LIN {X 0,Y 530.47,Z 630.938,A -85,B 0,C 180,E1 -4406.963,E2 -4406.963} C_VEL
LIN {X 0,Y 530.412,Z 632.682,A -85,B 0,C 180,E1 -4407.722,E2 -4407.722} C_VEL
LIN {X 0,Y 530.36,Z 633.93,A -85,B 0,C 180,E1 -4408.482,E2 -4408.482} C_VEL
LIN {X 0,Y 530.342,Z 634.707,A -85,B 0,C 180,E1 -4409.241,E2 -4409.241} C_VEL
LIN {X 0,Y 530.34,Z 635,A -85,B 0,C 180,E1 -4410,E2 -4410} C_VEL
LIN {X 0,Y 530.342,Z 634.706,A -85,B 0,C 180,E1 -4410.76,E2 -4410.76} C_VEL
LIN {X 0,Y 530.36,Z 633.928,A -85,B 0,C 180,E1 -4411.519,E2 -4411.519} C_VEL
LIN {X 0,Y 530.412,Z 632.679,A -85,B 0,C 180,E1 -4412.279,E2 -4412.279} C_VEL
LIN {X 0,Y 530.501,Z 629.785,A -85,B 0,C 180,E1 -4413.418,E2 -4413.418} C_VEL
LIN {X 0,Y 530.546,Z 627.147,A -85,B 0,C 180,E1 -4414.178,E2 -4414.178} C_VEL
LIN {X 0,Y 530.543,Z 621.984,A -85,B 0,C 180,E1 -4415.321,E2 -4415.321} C_VEL
LIN {X 0,Y 530.729,Z 616.44,A -85,B 0,C 180,E1 -4416.271,E2 -4416.271} C_VEL
LIN {X 0,Y 530.794,Z 609.432,A -85,B 0,C 180,E1 -4417.226,E2 -4417.226} C_VEL
LIN {X 0,Y 530.928,Z 601.415,A -85,B 0,C 180,E1 -4418.086,E2 -4418.086} C_VEL
LIN {X 0,Y 531.106,Z 593.759,A -85,B 0,C 180,E1 -4418.753,E2 -4418.753} C_VEL
LIN {X 0,Y 531.226,Z 585.716,A -85,B 0,C 180,E1 -4419.327,E2 -4419.327} C_VEL
LIN {X 0,Y 531.389,Z 577.382,A -85,B 0,C 180,E1 -4419.805,E2 -4419.805} C_VEL
LIN {X 0,Y 531.523,Z 568.876,A -85,B 0,C 180,E1 -4420.187,E2 -4420.187} C_VEL
LIN {X 0,Y 531.454,Z 560.399,A -85,B 0,C 180,E1 -4420.477,E2 -4420.477} C_VEL
LIN {X 0,Y 530.57,Z 553.301,A -85,B 0,C 180,E1 -4420.688,E2 -4420.688} C_VEL
LIN {X 0,Y 530.658,Z 544.2,A -85,B 0,C 180,E1 -4423.402,E2 -4423.402} C_VEL
LIN {X 0,Y 530.751,Z 534.941,A -85,B 0,C 180,E1 -4426.146,E2 -4426.146} C_VEL
LIN {X 0,Y 530.856,Z 525.622,A -85,B 0,C 180,E1 -4428.927,E2 -4428.927} C_VEL
LIN {X 0,Y 530.984,Z 515.377,A -85,B 0,C 180,E1 -4432.104,E2 -4432.104} C_VEL
LIN {X 0,Y 531.159,Z 506.089,A -85,B 0,C 180,E1 -4435.05,E2 -4435.05} C_VEL
LIN {X 0,Y 531.329,Z 497.227,A -85,B 0,C 180,E1 -4438.006,E2 -4438.006} C_VEL
LIN {X 0,Y 531.612,Z 488.788,A -85,B 0,C 180,E1 -4441.037,E2 -4441.037} C_VEL
LIN {X 0,Y 531.787,Z 484.27,A -85,B 0,C 180,E1 -4442.81,E2 -4442.81} C_VEL
LIN {X 0,Y 530.978,Z 479.161,A -85,B 0,C 180,E1 -4445.126,E2 -4445.126} C_VEL
LIN {X 0,Y 530.969,Z 479.161,A -85,B 0,C 180,E1 -4447.508,E2 -4447.508} C_VEL
LIN {X 0,Y 530.986,Z 479.159,A -85,B 0,C 180,E1 -4450.433,E2 -4450.433} C_VEL
LIN {X 0,Y 530.968,Z 479.162,A -85,B 0,C 180,E1 -4453.495,E2 -4453.495} C_VEL
LIN {X 0,Y 530.97,Z 479.161,A -85,B 0,C 180,E1 -4456.506,E2 -4456.506} C_VEL
LIN {X 0,Y 530.984,Z 479.159,A -85,B 0,C 180,E1 -4459.567,E2 -4459.567} C_VEL
LIN {X 0,Y 530.971,Z 479.159,A -85,B 0,C 180,E1 -4462.577,E2 -4462.577} C_VEL
LIN {X 0,Y 530.985,Z 479.156,A -85,B 0,C 180,E1 -4465.31,E2 -4465.31} C_VEL
LIN {X 0,Y 530.889,Z 479.172,A -85,B 0,C 180,E1 -4468.027,E2 -4468.027} C_VEL
LIN {X 0,Y 530.823,Z 481.04,A -85,B 0,C 180,E1 -4469.794,E2 -4469.794} C_VEL
LIN {X 0,Y 530.741,Z 484.422,A -85,B 0,C 180,E1 -4472.525,E2 -4472.525} C_VEL
LIN {X 0,Y 530.652,Z 487.475,A -85,B 0,C 180,E1 -4474.925,E2 -4474.925} C_VEL
LIN {X 0,Y 530.59,Z 490.671,A -85,B 0,C 180,E1 -4477.411,E2 -4477.411} C_VEL
LIN {X 0,Y 530.592,Z 494.26,A -85,B 0,C 180,E1 -4480.126,E2 -4480.126} C_VEL
LIN {X 0,Y 530.52,Z 498.183,A -85,B 0,C 180,E1 -4483.056,E2 -4483.056} C_VEL
LIN {X 0,Y 530.533,Z 501.331,A -85,B 0,C 180,E1 -4485.422,E2 -4485.422} C_VEL
LIN {X 0,Y 530.451,Z 505.76,A -85,B 0,C 180,E1 -4488.649,E2 -4488.649} C_VEL
LIN {X 0,Y 530.428,Z 506.855,A -85,B 0,C 180,E1 -4489.431,E2 -4489.431} C_VEL
LIN {X 0,Y 531.541,Z 516.565,A -85,B 0,C 180,E1 -4489.766,E2 -4489.766} C_VEL
LIN {X 0,Y 531.394,Z 526.519,A -85,B 0,C 180,E1 -4490.196,E2 -4490.196} C_VEL
LIN {X 0,Y 531.236,Z 535.019,A -85,B 0,C 180,E1 -4490.673,E2 -4490.673} C_VEL
LIN {X 0,Y 531.105,Z 543.186,A -85,B 0,C 180,E1 -4491.247,E2 -4491.247} C_VEL
LIN {X 0,Y 530.929,Z 550.939,A -85,B 0,C 180,E1 -4491.915,E2 -4491.915} C_VEL
LIN {X 0,Y 530.797,Z 559.04,A -85,B 0,C 180,E1 -4492.774,E2 -4492.774} C_VEL
LIN {X 0,Y 530.739,Z 566.143,A -85,B 0,C 180,E1 -4493.726,E2 -4493.726} C_VEL
LIN {X 0,Y 530.544,Z 571.76,A -85,B 0,C 180,E1 -4494.68,E2 -4494.68} C_VEL
LIN {X 0,Y 530.547,Z 576.97,A -85,B 0,C 180,E1 -4495.822,E2 -4495.822} C_VEL
LIN {X 0,Y 530.503,Z 579.65,A -85,B 0,C 180,E1 -4496.582,E2 -4496.582} C_VEL
LIN {X 0,Y 530.411,Z 582.584,A -85,B 0,C 180,E1 -4497.722,E2 -4497.722} C_VEL
LIN {X 0,Y 530.361,Z 583.871,A -85,B 0,C 180,E1 -4498.481,E2 -4498.481} C_VEL
LIN {X 0,Y 530.341,Z 584.687,A -85,B 0,C 180,E1 -4499.241,E2 -4499.241} C_VEL
LIN {X 0,Y 530.339,Z 584.997,A -85,B 0,C 180,E1 -4500,E2 -4500} C_VEL
LIN {X 0,Y 530.343,Z 584.725,A -85,B 0,C 180,E1 -4500.759,E2 -4500.759} C_VEL
LIN {X 0,Y 530.36,Z 583.986,A -85,B 0,C 180,E1 -4501.519,E2 -4501.519} C_VEL
LIN {X 0,Y 530.411,Z 582.776,A -85,B 0,C 180,E1 -4502.278,E2 -4502.278} C_VEL
LIN {X 0,Y 530.491,Z 579.923,A -85,B 0,C 180,E1 -4503.418,E2 -4503.418} C_VEL
LIN {X 0,Y 530.546,Z 577.328,A -85,B 0,C 180,E1 -4504.178,E2 -4504.178} C_VEL
LIN {X 0,Y 530.541,Z 572.214,A -85,B 0,C 180,E1 -4505.321,E2 -4505.321} C_VEL
LIN {X 0,Y 530.729,Z 566.748,A -85,B 0,C 180,E1 -4506.266,E2 -4506.266} C_VEL
LIN {X 0,Y 530.795,Z 559.812,A -85,B 0,C 180,E1 -4507.226,E2 -4507.226} C_VEL
LIN {X 0,Y 530.918,Z 551.89,A -85,B 0,C 180,E1 -4508.085,E2 -4508.085} C_VEL
LIN {X 0,Y 531.092,Z 544.335,A -85,B 0,C 180,E1 -4508.753,E2 -4508.753} C_VEL
LIN {X 0,Y 531.22,Z 536.423,A -85,B 0,C 180,E1 -4509.327,E2 -4509.327} C_VEL
LIN {X 0,Y 531.392,Z 528.262,A -85,B 0,C 180,E1 -4509.804,E2 -4509.804} C_VEL
LIN {X 0,Y 531.484,Z 520.02,A -85,B 0,C 180,E1 -4510.187,E2 -4510.187} C_VEL
LIN {X 0,Y 531.275,Z 513.221,A -85,B 0,C 180,E1 -4510.444,E2 -4510.444} C_VEL
LIN {X 0,Y 530.419,Z 506.574,A -85,B 0,C 180,E1 -4510.666,E2 -4510.666} C_VEL
LIN {X 0,Y 530.455,Z 502.979,A -85,B 0,C 180,E1 -4513.017,E2 -4513.017} C_VEL
LIN {X 0,Y 530.498,Z 499.448,A -85,B 0,C 180,E1 -4515.365,E2 -4515.365} C_VEL
LIN {X 0,Y 530.51,Z 495.947,A -85,B 0,C 180,E1 -4517.74,E2 -4517.74} C_VEL
LIN {X 0,Y 530.574,Z 492.447,A -85,B 0,C 180,E1 -4520.145,E2 -4520.145} C_VEL
LIN {X 0,Y 530.535,Z 488.732,A -85,B 0,C 180,E1 -4522.592,E2 -4522.592} C_VEL
LIN {X 0,Y 530.602,Z 485.059,A -85,B 0,C 180,E1 -4525.078,E2 -4525.078} C_VEL
LIN {X 0,Y 530.739,Z 481.892,A -85,B 0,C 180,E1 -4527.292,E2 -4527.292} C_VEL
LIN {X 0,Y 530.746,Z 488.059,A -85,B 0,C 180,E1 -4529.773,E2 -4529.773} C_VEL
LIN {X 0,Y 530.77,Z 494.522,A -85,B 0,C 180,E1 -4532.439,E2 -4532.439} C_VEL
LIN {X 0,Y 530.667,Z 500.16,A -85,B 0,C 180,E1 -4534.803,E2 -4534.803} C_VEL
LIN {X 0,Y 530.626,Z 506.621,A -85,B 0,C 180,E1 -4537.536,E2 -4537.536} C_VEL
LIN {X 0,Y 530.597,Z 511.429,A -85,B 0,C 180,E1 -4539.542,E2 -4539.542} C_VEL
LIN {X 0,Y 529.942,Z 512.958,A -85,B 0,C 180,E1 -4540.154,E2 -4540.154} C_VEL
LIN {X 0,Y 527.033,Z 515.502,A -85,B 0,C 180,E1 -4541.145,E2 -4541.145} C_VEL
LIN {X 0,Y 524.569,Z 517.514,A -85,B 0,C 180,E1 -4541.944,E2 -4541.944} C_VEL
LIN {X 0,Y 523.523,Z 518.992,A -85,B 0,C 180,E1 -4542.563,E2 -4542.563} C_VEL
LIN {X 0,Y 523.447,Z 519.474,A -85,B 0,C 180,E1 -4542.773,E2 -4542.773} C_VEL
LIN {X 0,Y 523.418,Z 525.143,A -85,B 0,C 180,E1 -4545.254,E2 -4545.254} C_VEL
LIN {X 0,Y 524.584,Z 535.182,A -85,B 0,C 180,E1 -4545.573,E2 -4545.573} C_VEL
LIN {X 0,Y 524.442,Z 546.72,A -85,B 0,C 180,E1 -4546.064,E2 -4546.064} C_VEL
LIN {X 0,Y 524.216,Z 556.215,A -85,B 0,C 180,E1 -4546.615,E2 -4546.615} C_VEL
LIN {X 0,Y 524.055,Z 564.577,A -85,B 0,C 180,E1 -4547.23,E2 -4547.23} C_VEL
LIN {X 0,Y 523.854,Z 572.859,A -85,B 0,C 180,E1 -4547.987,E2 -4547.987} C_VEL
LIN {X 0,Y 523.695,Z 579.437,A -85,B 0,C 180,E1 -4548.722,E2 -4548.722} C_VEL
LIN {X 0,Y 523.595,Z 584.439,A -85,B 0,C 180,E1 -4549.383,E2 -4549.383} C_VEL
LIN {X 0,Y 523.513,Z 590.665,A -85,B 0,C 180,E1 -4550.399,E2 -4550.399} C_VEL
LIN {X 0,Y 523.446,Z 594.425,A -85,B 0,C 180,E1 -4551.145,E2 -4551.145} C_VEL
LIN {X 0,Y 523.416,Z 597.403,A -85,B 0,C 180,E1 -4551.855,E2 -4551.855} C_VEL
LIN {X 0,Y 523.337,Z 600.555,A -85,B 0,C 180,E1 -4552.82,E2 -4552.82} C_VEL
LIN {X 0,Y 523.282,Z 602.795,A -85,B 0,C 180,E1 -4553.775,E2 -4553.775} C_VEL
LIN {X 0,Y 523.279,Z 604.553,A -85,B 0,C 180,E1 -4555.012,E2 -4555.012} C_VEL
LIN {X 0,Y 523.279,Z 604.883,A -85,B 0,C 180,E1 -4556.377,E2 -4556.377} C_VEL
LIN {X 0,Y 523.278,Z 603.641,A -85,B 0,C 180,E1 -4557.794,E2 -4557.794} C_VEL
LIN {X 0,Y 523.31,Z 602.57,A -85,B 0,C 180,E1 -4558.414,E2 -4558.414} C_VEL
LIN {X 0,Y 523.392,Z 600.399,A -85,B 0,C 180,E1 -4559.319,E2 -4559.319} C_VEL
LIN {X 0,Y 523.42,Z 596.195,A -85,B 0,C 180,E1 -4560.525,E2 -4560.525} C_VEL
LIN {X 0,Y 523.454,Z 592.668,A -85,B 0,C 180,E1 -4561.315,E2 -4561.315} C_VEL
LIN {X 0,Y 523.556,Z 587.76,A -85,B 0,C 180,E1 -4562.201,E2 -4562.201} C_VEL
LIN {X 0,Y 523.668,Z 581.842,A -85,B 0,C 180,E1 -4563.067,E2 -4563.067} C_VEL
LIN {X 0,Y 523.803,Z 574.832,A -85,B 0,C 180,E1 -4563.9,E2 -4563.9} C_VEL
LIN {X 0,Y 523.945,Z 567.889,A -85,B 0,C 180,E1 -4564.581,E2 -4564.581} C_VEL
LIN {X 0,Y 524.142,Z 559.814,A -85,B 0,C 180,E1 -4565.227,E2 -4565.227} C_VEL
LIN {X 0,Y 524.261,Z 550.824,A -85,B 0,C 180,E1 -4565.803,E2 -4565.803} C_VEL
LIN {X 0,Y 524.478,Z 541.798,A -85,B 0,C 180,E1 -4566.253,E2 -4566.253} C_VEL
LIN {X 0,Y 524.415,Z 533.272,A -85,B 0,C 180,E1 -4566.581,E2 -4566.581} C_VEL
LIN {X 0,Y 523.368,Z 525.332,A -85,B 0,C 180,E1 -4566.846,E2 -4566.846} C_VEL
LIN {X 0,Y 523.456,Z 518.488,A -85,B 0,C 180,E1 -4570.023,E2 -4570.023} C_VEL
LIN {X 0,Y 523.489,Z 512.468,A -85,B 0,C 180,E1 -4572.821,E2 -4572.821} C_VEL
LIN {X 0,Y 523.565,Z 505.401,A -85,B 0,C 180,E1 -4576.017,E2 -4576.017} C_VEL
LIN {X 0,Y 523.665,Z 498.515,A -85,B 0,C 180,E1 -4579.17,E2 -4579.17} C_VEL
LIN {X 0,Y 523.664,Z 491.614,A -85,B 0,C 180,E1 -4582.287,E2 -4582.287} C_VEL
LIN {X 0,Y 523.761,Z 484.698,A -85,B 0,C 180,E1 -4585.382,E2 -4585.382} C_VEL
LIN {X 0,Y 523.697,Z 480.067,A -85,B 0,C 180,E1 -4587.5,E2 -4587.5} C_VEL
LIN {X 0,Y 524.123,Z 480.013,A -85,B 0,C 180,E1 -4589.231,E2 -4589.231} C_VEL
LIN {X 0,Y 524.115,Z 480.013,A -85,B 0,C 180,E1 -4592.305,E2 -4592.305} C_VEL
LIN {X 0,Y 524.087,Z 480.017,A -85,B 0,C 180,E1 -4595.386,E2 -4595.386} C_VEL
LIN {X 0,Y 524.003,Z 480.028,A -85,B 0,C 180,E1 -4598.484,E2 -4598.484} C_VEL
LIN {X 0,Y 524.004,Z 480.026,A -85,B 0,C 180,E1 -4601.739,E2 -4601.739} C_VEL
LIN {X 0,Y 523.995,Z 480.027,A -85,B 0,C 180,E1 -4605.052,E2 -4605.052} C_VEL
LIN {X 0,Y 523.966,Z 480.032,A -85,B 0,C 180,E1 -4607.968,E2 -4607.968} C_VEL
LIN {X 0,Y 523.973,Z 480.032,A -85,B 0,C 180,E1 -4610.41,E2 -4610.41} C_VEL
LIN {X 0,Y 523.918,Z 480.039,A -85,B 0,C 180,E1 -4612.893,E2 -4612.893} C_VEL
LIN {X 0,Y 523.956,Z 480.034,A -85,B 0,C 180,E1 -4615.418,E2 -4615.418} C_VEL
LIN {X 0,Y 523.971,Z 480.032,A -85,B 0,C 180,E1 -4617.998,E2 -4617.998} C_VEL
LIN {X 0,Y 523.953,Z 480.033,A -85,B 0,C 180,E1 -4620.856,E2 -4620.856} C_VEL
LIN {X 0,Y 523.961,Z 480.034,A -85,B 0,C 180,E1 -4623.735,E2 -4623.735} C_VEL
LIN {X 0,Y 523.923,Z 480.037,A -85,B 0,C 180,E1 -4626.404,E2 -4626.404} C_VEL
LIN {X 0,Y 523.922,Z 480.036,A -85,B 0,C 180,E1 -4629.084,E2 -4629.084} C_VEL
LIN {X 0,Y 523.953,Z 480.034,A -85,B 0,C 180,E1 -4632.118,E2 -4632.118} C_VEL
LIN {X 0,Y 523.955,Z 480.033,A -85,B 0,C 180,E1 -4635.308,E2 -4635.308} C_VEL
LIN {X 0,Y 523.973,Z 480.031,A -85,B 0,C 180,E1 -4638.687,E2 -4638.687} C_VEL
LIN {X 0,Y 523.952,Z 480.033,A -85,B 0,C 180,E1 -4641.075,E2 -4641.075} C_VEL
LIN {X 0,Y 523.898,Z 480.042,A -85,B 0,C 180,E1 -4643.825,E2 -4643.825} C_VEL
LIN {X 0,Y 523.94,Z 480.034,A -85,B 0,C 180,E1 -4646.635,E2 -4646.635} C_VEL
LIN {X 0,Y 523.955,Z 480.032,A -85,B 0,C 180,E1 -4649.356,E2 -4649.356} C_VEL
LIN {X 0,Y 523.979,Z 480.03,A -85,B 0,C 180,E1 -4652.28,E2 -4652.28} C_VEL
LIN {X 0,Y 523.954,Z 480.032,A -85,B 0,C 180,E1 -4654.581,E2 -4654.581} C_VEL
LIN {X 0,Y 523.915,Z 480.037,A -85,B 0,C 180,E1 -4657.107,E2 -4657.107} C_VEL
LIN {X 0,Y 523.978,Z 480.03,A -85,B 0,C 180,E1 -4659.865,E2 -4659.865} C_VEL
LIN {X 0,Y 523.965,Z 480.032,A -85,B 0,C 180,E1 -4662.837,E2 -4662.837} C_VEL
LIN {X 0,Y 523.975,Z 480.031,A -85,B 0,C 180,E1 -4665.236,E2 -4665.236} C_VEL
LIN {X 0,Y 524.013,Z 480.028,A -85,B 0,C 180,E1 -4668.394,E2 -4668.394} C_VEL
LIN {X 0,Y 524.003,Z 480.027,A -85,B 0,C 180,E1 -4671.516,E2 -4671.516} C_VEL
LIN {X 0,Y 524.081,Z 480.017,A -85,B 0,C 180,E1 -4674.614,E2 -4674.614} C_VEL
LIN {X 0,Y 524.112,Z 480.014,A -85,B 0,C 180,E1 -4677.694,E2 -4677.694} C_VEL
LIN {X 0,Y 524.122,Z 480.011,A -85,B 0,C 180,E1 -4680.768,E2 -4680.768} C_VEL
LIN {X 0,Y 524.074,Z 480.018,A -85,B 0,C 180,E1 -4683.075,E2 -4683.075} C_VEL
LIN {X 0,Y 524.046,Z 480.024,A -85,B 0,C 180,E1 -4686.159,E2 -4686.159} C_VEL
LIN {X 0,Y 523.999,Z 480.027,A -85,B 0,C 180,E1 -4689.262,E2 -4689.262} C_VEL
LIN {X 0,Y 524.001,Z 480.027,A -85,B 0,C 180,E1 -4691.74,E2 -4691.74} C_VEL
LIN {X 0,Y 523.99,Z 480.028,A -85,B 0,C 180,E1 -4695.052,E2 -4695.052} C_VEL
LIN {X 0,Y 523.962,Z 480.034,A -85,B 0,C 180,E1 -4697.969,E2 -4697.969} C_VEL
LIN {X 0,Y 523.97,Z 480.032,A -85,B 0,C 180,E1 -4700.41,E2 -4700.41} C_VEL
LIN {X 0,Y 523.915,Z 480.039,A -85,B 0,C 180,E1 -4702.893,E2 -4702.893} C_VEL
LIN {X 0,Y 523.951,Z 480.034,A -85,B 0,C 180,E1 -4705.419,E2 -4705.419} C_VEL
LIN {X 0,Y 523.967,Z 480.031,A -85,B 0,C 180,E1 -4707.999,E2 -4707.999} C_VEL
LIN {X 0,Y 523.951,Z 480.033,A -85,B 0,C 180,E1 -4710.857,E2 -4710.857} C_VEL
LIN {X 0,Y 523.959,Z 480.033,A -85,B 0,C 180,E1 -4713.735,E2 -4713.735} C_VEL
LIN {X 0,Y 523.921,Z 480.036,A -85,B 0,C 180,E1 -4716.405,E2 -4716.405} C_VEL
LIN {X 0,Y 523.918,Z 480.038,A -85,B 0,C 180,E1 -4719.085,E2 -4719.085} C_VEL
LIN {X 0,Y 523.956,Z 480.032,A -85,B 0,C 180,E1 -4722.118,E2 -4722.118} C_VEL
LIN {X 0,Y 523.953,Z 480.035,A -85,B 0,C 180,E1 -4725.309,E2 -4725.309} C_VEL
LIN {X 0,Y 523.971,Z 480.032,A -85,B 0,C 180,E1 -4728.688,E2 -4728.688} C_VEL
LIN {X 0,Y 523.952,Z 480.035,A -85,B 0,C 180,E1 -4731.076,E2 -4731.076} C_VEL
LIN {X 0,Y 523.927,Z 480.037,A -85,B 0,C 180,E1 -4733.828,E2 -4733.828} C_VEL
LIN {X 0,Y 523.978,Z 480.097,A -85,B 0,C 180,E1 -4736.868,E2 -4736.868} C_VEL
LIN {X 0,Y 524.761,Z 484.749,A -85,B 0,C 180,E1 -4738.513,E2 -4738.513} C_VEL
LIN {X 0,Y 524.676,Z 490.829,A -85,B 0,C 180,E1 -4740.537,E2 -4740.537} C_VEL
LIN {X 0,Y 524.437,Z 499.476,A -85,B 0,C 180,E1 -4743.325,E2 -4743.325} C_VEL
LIN {X 0,Y 524.185,Z 508.922,A -85,B 0,C 180,E1 -4746.283,E2 -4746.283} C_VEL
LIN {X 0,Y 524.034,Z 518.43,A -85,B 0,C 180,E1 -4749.182,E2 -4749.182} C_VEL
LIN {X 0,Y 523.812,Z 528.83,A -85,B 0,C 180,E1 -4752.29,E2 -4752.29} C_VEL
LIN {X 0,Y 523.702,Z 539.019,A -85,B 0,C 180,E1 -4755.228,E2 -4755.228} C_VEL
LIN {X 0,Y 523.603,Z 550.38,A -85,B 0,C 180,E1 -4758.473,E2 -4758.473} C_VEL
LIN {X 0,Y 523.549,Z 552.826,A -85,B 0,C 180,E1 -4759.168,E2 -4759.168} C_VEL
LIN {X 0,Y 524.574,Z 563.488,A -85,B 0,C 180,E1 -4759.483,E2 -4759.483} C_VEL
LIN {X 0,Y 524.423,Z 575.323,A -85,B 0,C 180,E1 -4759.967,E2 -4759.967} C_VEL
LIN {X 0,Y 524.232,Z 584.068,A -85,B 0,C 180,E1 -4760.451,E2 -4760.451} C_VEL
LIN {X 0,Y 524.122,Z 592.427,A -85,B 0,C 180,E1 -4761.033,E2 -4761.033} C_VEL
LIN {X 0,Y 523.923,Z 600.332,A -85,B 0,C 180,E1 -4761.709,E2 -4761.709} C_VEL
LIN {X 0,Y 523.757,Z 607.725,A -85,B 0,C 180,E1 -4762.483,E2 -4762.483} C_VEL
LIN {X 0,Y 523.659,Z 615.797,A -85,B 0,C 180,E1 -4763.54,E2 -4763.54} C_VEL
LIN {X 0,Y 523.485,Z 621.991,A -85,B 0,C 180,E1 -4764.608,E2 -4764.608} C_VEL
LIN {X 0,Y 523.472,Z 627.151,A -85,B 0,C 180,E1 -4765.766,E2 -4765.766} C_VEL
LIN {X 0,Y 523.381,Z 630.939,A -85,B 0,C 180,E1 -4766.921,E2 -4766.921} C_VEL
LIN {X 0,Y 523.336,Z 632.681,A -85,B 0,C 180,E1 -4767.691,E2 -4767.691} C_VEL
LIN {X 0,Y 523.273,Z 633.929,A -85,B 0,C 180,E1 -4768.461,E2 -4768.461} C_VEL
LIN {X 0,Y 523.248,Z 634.706,A -85,B 0,C 180,E1 -4769.231,E2 -4769.231} C_VEL
LIN {X 0,Y 523.244,Z 635,A -85,B 0,C 180,E1 -4770,E2 -4770} C_VEL
LIN {X 0,Y 523.248,Z 634.705,A -85,B 0,C 180,E1 -4770.77,E2 -4770.77} C_VEL
LIN {X 0,Y 523.273,Z 633.927,A -85,B 0,C 180,E1 -4771.54,E2 -4771.54} C_VEL
LIN {X 0,Y 523.336,Z 632.678,A -85,B 0,C 180,E1 -4772.309,E2 -4772.309} C_VEL
LIN {X 0,Y 523.413,Z 629.785,A -85,B 0,C 180,E1 -4773.464,E2 -4773.464} C_VEL
LIN {X 0,Y 523.47,Z 627.147,A -85,B 0,C 180,E1 -4774.235,E2 -4774.235} C_VEL
LIN {X 0,Y 523.485,Z 621.984,A -85,B 0,C 180,E1 -4775.393,E2 -4775.393} C_VEL
LIN {X 0,Y 523.668,Z 615.737,A -85,B 0,C 180,E1 -4776.469,E2 -4776.469} C_VEL
LIN {X 0,Y 523.758,Z 607.72,A -85,B 0,C 180,E1 -4777.518,E2 -4777.518} C_VEL
LIN {X 0,Y 523.924,Z 600.325,A -85,B 0,C 180,E1 -4778.291,E2 -4778.291} C_VEL
LIN {X 0,Y 524.123,Z 592.401,A -85,B 0,C 180,E1 -4778.968,E2 -4778.968} C_VEL
LIN {X 0,Y 524.243,Z 584.023,A -85,B 0,C 180,E1 -4779.55,E2 -4779.55} C_VEL
LIN {X 0,Y 524.459,Z 573.336,A -85,B 0,C 180,E1 -4780.13,E2 -4780.13} C_VEL
LIN {X 0,Y 524.584,Z 562.538,A -85,B 0,C 180,E1 -4780.542,E2 -4780.542} C_VEL
LIN {X 0,Y 523.502,Z 553.04,A -85,B 0,C 180,E1 -4780.834,E2 -4780.834} C_VEL
LIN {X 0,Y 523.601,Z 542.52,A -85,B 0,C 180,E1 -4783.982,E2 -4783.982} C_VEL
LIN {X 0,Y 523.688,Z 533.247,A -85,B 0,C 180,E1 -4786.771,E2 -4786.771} C_VEL
LIN {X 0,Y 523.834,Z 524.034,A -85,B 0,C 180,E1 -4789.598,E2 -4789.598} C_VEL
LIN {X 0,Y 523.992,Z 513.633,A -85,B 0,C 180,E1 -4792.89,E2 -4792.89} C_VEL
LIN {X 0,Y 524.182,Z 503.917,A -85,B 0,C 180,E1 -4796.064,E2 -4796.064} C_VEL
LIN {X 0,Y 524.39,Z 495.936,A -85,B 0,C 180,E1 -4798.848,E2 -4798.848} C_VEL
LIN {X 0,Y 524.683,Z 488.876,A -85,B 0,C 180,E1 -4801.493,E2 -4801.493} C_VEL
LIN {X 0,Y 524.82,Z 486.443,A -85,B 0,C 180,E1 -4802.473,E2 -4802.473} C_VEL
LIN {X 0,Y 524.412,Z 482.418,A -85,B 0,C 180,E1 -4804.255,E2 -4804.255} C_VEL
LIN {X 0,Y 523.936,Z 480.038,A -85,B 0,C 180,E1 -4805.461,E2 -4805.461} C_VEL
LIN {X 0,Y 523.919,Z 480.039,A -85,B 0,C 180,E1 -4808.102,E2 -4808.102} C_VEL
LIN {X 0,Y 523.944,Z 480.034,A -85,B 0,C 180,E1 -4811.092,E2 -4811.092} C_VEL
LIN {X 0,Y 523.944,Z 480.033,A -85,B 0,C 180,E1 -4814.228,E2 -4814.228} C_VEL
LIN {X 0,Y 523.928,Z 480.038,A -85,B 0,C 180,E1 -4816.834,E2 -4816.834} C_VEL
LIN {X 0,Y 523.944,Z 480.033,A -85,B 0,C 180,E1 -4818.908,E2 -4818.908} C_VEL
LIN {X 0,Y 523.918,Z 480.037,A -85,B 0,C 180,E1 -4821.898,E2 -4821.898} C_VEL
LIN {X 0,Y 523.927,Z 480.038,A -85,B 0,C 180,E1 -4824.911,E2 -4824.911} C_VEL
LIN {X 0,Y 523.871,Z 480.046,A -85,B 0,C 180,E1 -4827.692,E2 -4827.692} C_VEL
LIN {X 0,Y 523.819,Z 480.37,A -85,B 0,C 180,E1 -4828.449,E2 -4828.449} C_VEL
LIN {X 0,Y 523.713,Z 483.539,A -85,B 0,C 180,E1 -4831.112,E2 -4831.112} C_VEL
LIN {X 0,Y 523.654,Z 487.162,A -85,B 0,C 180,E1 -4834.055,E2 -4834.055} C_VEL
LIN {X 0,Y 523.584,Z 489.932,A -85,B 0,C 180,E1 -4836.254,E2 -4836.254} C_VEL
LIN {X 0,Y 523.532,Z 494.212,A -85,B 0,C 180,E1 -4839.572,E2 -4839.572} C_VEL
LIN {X 0,Y 523.445,Z 498.554,A -85,B 0,C 180,E1 -4842.82,E2 -4842.82} C_VEL
LIN {X 0,Y 523.465,Z 501.697,A -85,B 0,C 180,E1 -4845.221,E2 -4845.221} C_VEL
LIN {X 0,Y 523.399,Z 506.246,A -85,B 0,C 180,E1 -4848.586,E2 -4848.586} C_VEL
LIN {X 0,Y 523.388,Z 507.452,A -85,B 0,C 180,E1 -4849.311,E2 -4849.311} C_VEL
LIN {X 0,Y 524.547,Z 516.773,A -85,B 0,C 180,E1 -4849.628,E2 -4849.628} C_VEL
LIN {X 0,Y 524.405,Z 526.74,A -85,B 0,C 180,E1 -4850.064,E2 -4850.064} C_VEL
LIN {X 0,Y 524.238,Z 535.245,A -85,B 0,C 180,E1 -4850.548,E2 -4850.548} C_VEL
LIN {X 0,Y 524.094,Z 543.404,A -85,B 0,C 180,E1 -4851.129,E2 -4851.129} C_VEL
LIN {X 0,Y 523.918,Z 551.144,A -85,B 0,C 180,E1 -4851.806,E2 -4851.806} C_VEL
LIN {X 0,Y 523.761,Z 557.531,A -85,B 0,C 180,E1 -4852.483,E2 -4852.483} C_VEL
LIN {X 0,Y 523.672,Z 563.785,A -85,B 0,C 180,E1 -4853.281,E2 -4853.281} C_VEL
LIN {X 0,Y 523.547,Z 570.93,A -85,B 0,C 180,E1 -4854.415,E2 -4854.415} C_VEL
LIN {X 0,Y 523.422,Z 575.568,A -85,B 0,C 180,E1 -4855.379,E2 -4855.379} C_VEL
LIN {X 0,Y 523.459,Z 578.555,A -85,B 0,C 180,E1 -4856.151,E2 -4856.151} C_VEL
LIN {X 0,Y 523.384,Z 580.875,A -85,B 0,C 180,E1 -4856.921,E2 -4856.921} C_VEL
LIN {X 0,Y 523.336,Z 582.646,A -85,B 0,C 180,E1 -4857.691,E2 -4857.691} C_VEL
LIN {X 0,Y 523.275,Z 583.925,A -85,B 0,C 180,E1 -4858.461,E2 -4858.461} C_VEL
LIN {X 0,Y 523.248,Z 584.735,A -85,B 0,C 180,E1 -4859.23,E2 -4859.23} C_VEL
LIN {X 0,Y 523.243,Z 585.042,A -85,B 0,C 180,E1 -4860,E2 -4860} C_VEL
LIN {X 0,Y 523.249,Z 584.771,A -85,B 0,C 180,E1 -4860.77,E2 -4860.77} C_VEL
LIN {X 0,Y 523.274,Z 584.035,A -85,B 0,C 180,E1 -4861.539,E2 -4861.539} C_VEL
LIN {X 0,Y 523.335,Z 582.831,A -85,B 0,C 180,E1 -4862.309,E2 -4862.309} C_VEL
LIN {X 0,Y 523.404,Z 579.994,A -85,B 0,C 180,E1 -4863.464,E2 -4863.464} C_VEL
LIN {X 0,Y 523.469,Z 577.412,A -85,B 0,C 180,E1 -4864.235,E2 -4864.235} C_VEL
LIN {X 0,Y 523.485,Z 572.326,A -85,B 0,C 180,E1 -4865.393,E2 -4865.393} C_VEL
LIN {X 0,Y 523.643,Z 568.01,A -85,B 0,C 180,E1 -4866.164,E2 -4866.164} C_VEL
LIN {X 0,Y 523.704,Z 561.42,A -85,B 0,C 180,E1 -4867.131,E2 -4867.131} C_VEL
LIN {X 0,Y 523.853,Z 553.062,A -85,B 0,C 180,E1 -4868.098,E2 -4868.098} C_VEL
LIN {X 0,Y 524.089,Z 544.491,A -85,B 0,C 180,E1 -4868.871,E2 -4868.871} C_VEL
LIN {X 0,Y 524.232,Z 536.576,A -85,B 0,C 180,E1 -4869.452,E2 -4869.452} C_VEL
LIN {X 0,Y 524.408,Z 528.402,A -85,B 0,C 180,E1 -4869.936,E2 -4869.936} C_VEL
LIN {X 0,Y 524.507,Z 520.13,A -85,B 0,C 180,E1 -4870.324,E2 -4870.324} C_VEL
LIN {X 0,Y 524.461,Z 515.259,A -85,B 0,C 180,E1 -4870.52,E2 -4870.52} C_VEL
LIN {X 0,Y 523.353,Z 506.81,A -85,B 0,C 180,E1 -4870.812,E2 -4870.812} C_VEL
LIN {X 0,Y 523.365,Z 503.202,A -85,B 0,C 180,E1 -4873.196,E2 -4873.196} C_VEL
LIN {X 0,Y 523.41,Z 499.674,A -85,B 0,C 180,E1 -4875.578,E2 -4875.578} C_VEL
LIN {X 0,Y 523.423,Z 496.175,A -85,B 0,C 180,E1 -4877.988,E2 -4877.988} C_VEL
LIN {X 0,Y 523.482,Z 492.502,A -85,B 0,C 180,E1 -4880.43,E2 -4880.43} C_VEL
LIN {X 0,Y 523.539,Z 487.616,A -85,B 0,C 180,E1 -4883.748,E2 -4883.748} C_VEL
LIN {X 0,Y 523.567,Z 483.933,A -85,B 0,C 180,E1 -4886.294,E2 -4886.294} C_VEL
LIN {X 0,Y 523.693,Z 482.66,A -85,B 0,C 180,E1 -4887.311,E2 -4887.311} C_VEL
LIN {X 0,Y 523.666,Z 488.633,A -85,B 0,C 180,E1 -4889.773,E2 -4889.773} C_VEL
LIN {X 0,Y 523.699,Z 495.221,A -85,B 0,C 180,E1 -4892.466,E2 -4892.466} C_VEL
LIN {X 0,Y 523.58,Z 501.866,A -85,B 0,C 180,E1 -4895.253,E2 -4895.253} C_VEL
LIN {X 0,Y 523.551,Z 508.631,A -85,B 0,C 180,E1 -4898.133,E2 -4898.133} C_VEL
LIN {X 0,Y 523.494,Z 514.554,A -85,B 0,C 180,E1 -4900.626,E2 -4900.626} C_VEL
LIN {X 0,Y 523.447,Z 519.474,A -85,B 0,C 180,E1 -4902.773,E2 -4902.773} C_VEL
LIN {X 0,Y 522.776,Z 520.466,A -85,B 0,C 180,E1 -4903.188,E2 -4903.188} C_VEL
LIN {X 0,Y 519.907,Z 522.135,A -85,B 0,C 180,E1 -4903.832,E2 -4903.832} C_VEL
LIN {X 0,Y 517.019,Z 523.808,A -85,B 0,C 180,E1 -4904.483,E2 -4904.483} C_VEL
LIN {X 0,Y 516.338,Z 524.809,A -85,B 0,C 180,E1 -4904.906,E2 -4904.906} C_VEL
LIN {X 0,Y 516.337,Z 525.264,A -85,B 0,C 180,E1 -4905.107,E2 -4905.107} C_VEL
LIN {X 0,Y 517.61,Z 535.802,A -85,B 0,C 180,E1 -4905.449,E2 -4905.449} C_VEL
LIN {X 0,Y 517.457,Z 546.907,A -85,B 0,C 180,E1 -4905.929,E2 -4905.929} C_VEL
LIN {X 0,Y 517.195,Z 557.056,A -85,B 0,C 180,E1 -4906.533,E2 -4906.533} C_VEL
LIN {X 0,Y 517.005,Z 565.603,A -85,B 0,C 180,E1 -4907.181,E2 -4907.181} C_VEL
LIN {X 0,Y 516.81,Z 573.784,A -85,B 0,C 180,E1 -4907.952,E2 -4907.952} C_VEL
LIN {X 0,Y 516.607,Z 582.402,A -85,B 0,C 180,E1 -4908.974,E2 -4908.974} C_VEL
LIN {X 0,Y 516.5,Z 588.772,A -85,B 0,C 180,E1 -4909.942,E2 -4909.942} C_VEL
LIN {X 0,Y 516.384,Z 593.7,A -85,B 0,C 180,E1 -4910.875,E2 -4910.875} C_VEL
LIN {X 0,Y 516.301,Z 598.767,A -85,B 0,C 180,E1 -4912.14,E2 -4912.14} C_VEL
LIN {X 0,Y 516.252,Z 601.794,A -85,B 0,C 180,E1 -4913.202,E2 -4913.202} C_VEL
LIN {X 0,Y 516.167,Z 603.688,A -85,B 0,C 180,E1 -4914.163,E2 -4914.163} C_VEL
LIN {X 0,Y 516.205,Z 604.805,A -85,B 0,C 180,E1 -4915.122,E2 -4915.122} C_VEL
LIN {X 0,Y 516.178,Z 605.15,A -85,B 0,C 180,E1 -4916.155,E2 -4916.155} C_VEL
LIN {X 0,Y 516.175,Z 604.788,A -85,B 0,C 180,E1 -4917.001,E2 -4917.001} C_VEL
LIN {X 0,Y 516.192,Z 603.684,A -85,B 0,C 180,E1 -4917.927,E2 -4917.927} C_VEL
LIN {X 0,Y 516.298,Z 600.455,A -85,B 0,C 180,E1 -4919.407,E2 -4919.407} C_VEL
LIN {X 0,Y 516.339,Z 596.391,A -85,B 0,C 180,E1 -4920.589,E2 -4920.589} C_VEL
LIN {X 0,Y 516.381,Z 592.009,A -85,B 0,C 180,E1 -4921.552,E2 -4921.552} C_VEL
LIN {X 0,Y 516.542,Z 586.925,A -85,B 0,C 180,E1 -4922.445,E2 -4922.445} C_VEL
LIN {X 0,Y 516.657,Z 580.74,A -85,B 0,C 180,E1 -4923.327,E2 -4923.327} C_VEL
LIN {X 0,Y 516.82,Z 573.128,A -85,B 0,C 180,E1 -4924.205,E2 -4924.205} C_VEL
LIN {X 0,Y 517.046,Z 564.852,A -85,B 0,C 180,E1 -4924.971,E2 -4924.971} C_VEL
LIN {X 0,Y 517.257,Z 554.958,A -85,B 0,C 180,E1 -4925.7,E2 -4925.7} C_VEL
LIN {X 0,Y 517.474,Z 543.414,A -85,B 0,C 180,E1 -4926.328,E2 -4926.328} C_VEL
LIN {X 0,Y 517.458,Z 534.183,A -85,B 0,C 180,E1 -4926.698,E2 -4926.698} C_VEL
LIN {X 0,Y 516.287,Z 525.478,A -85,B 0,C 180,E1 -4926.987,E2 -4926.987} C_VEL
LIN {X 0,Y 516.383,Z 518.797,A -85,B 0,C 180,E1 -4930.107,E2 -4930.107} C_VEL
LIN {X 0,Y 516.42,Z 513.516,A -85,B 0,C 180,E1 -4932.578,E2 -4932.578} C_VEL
LIN {X 0,Y 516.502,Z 506.434,A -85,B 0,C 180,E1 -4935.822,E2 -4935.822} C_VEL
LIN {X 0,Y 516.586,Z 499.466,A -85,B 0,C 180,E1 -4939.02,E2 -4939.02} C_VEL
LIN {X 0,Y 516.603,Z 492.53,A -85,B 0,C 180,E1 -4942.181,E2 -4942.181} C_VEL
LIN {X 0,Y 516.694,Z 485.555,A -85,B 0,C 180,E1 -4945.318,E2 -4945.318} C_VEL
LIN {X 0,Y 516.626,Z 480.948,A -85,B 0,C 180,E1 -4947.466,E2 -4947.466} C_VEL
LIN {X 0,Y 517.092,Z 480.889,A -85,B 0,C 180,E1 -4949.221,E2 -4949.221} C_VEL
LIN {X 0,Y 517.087,Z 480.888,A -85,B 0,C 180,E1 -4952.336,E2 -4952.336} C_VEL
LIN {X 0,Y 517.015,Z 480.898,A -85,B 0,C 180,E1 -4956.243,E2 -4956.243} C_VEL
LIN {X 0,Y 516.947,Z 480.904,A -85,B 0,C 180,E1 -4959.389,E2 -4959.389} C_VEL
LIN {X 0,Y 516.954,Z 480.905,A -85,B 0,C 180,E1 -4961.807,E2 -4961.807} C_VEL
LIN {X 0,Y 516.948,Z 480.904,A -85,B 0,C 180,E1 -4965.147,E2 -4965.147} C_VEL
LIN {X 0,Y 516.927,Z 480.911,A -85,B 0,C 180,E1 -4968.222,E2 -4968.222} C_VEL
LIN {X 0,Y 516.913,Z 480.911,A -85,B 0,C 180,E1 -4970.701,E2 -4970.701} C_VEL
LIN {X 0,Y 516.912,Z 480.912,A -85,B 0,C 180,E1 -4974.071,E2 -4974.071} C_VEL
LIN {X 0,Y 516.929,Z 480.908,A -85,B 0,C 180,E1 -4976.657,E2 -4976.657} C_VEL
LIN {X 0,Y 516.92,Z 480.908,A -85,B 0,C 180,E1 -4979.525,E2 -4979.525} C_VEL
LIN {X 0,Y 516.901,Z 480.912,A -85,B 0,C 180,E1 -4982.544,E2 -4982.544} C_VEL
LIN {X 0,Y 516.883,Z 480.913,A -85,B 0,C 180,E1 -4985.332,E2 -4985.332} C_VEL
LIN {X 0,Y 516.881,Z 480.914,A -85,B 0,C 180,E1 -4987.943,E2 -4987.943} C_VEL
LIN {X 0,Y 516.883,Z 480.915,A -85,B 0,C 180,E1 -4990.741,E2 -4990.741} C_VEL
LIN {X 0,Y 516.903,Z 480.912,A -85,B 0,C 180,E1 -4992.829,E2 -4992.829} C_VEL
LIN {X 0,Y 516.921,Z 480.908,A -85,B 0,C 180,E1 -4995.01,E2 -4995.01} C_VEL
LIN {X 0,Y 516.923,Z 480.909,A -85,B 0,C 180,E1 -4998.397,E2 -4998.397} C_VEL
LIN {X 0,Y 516.905,Z 480.912,A -85,B 0,C 180,E1 -5001.286,E2 -5001.286} C_VEL
LIN {X 0,Y 516.869,Z 480.915,A -85,B 0,C 180,E1 -5004.219,E2 -5004.219} C_VEL
LIN {X 0,Y 516.896,Z 480.912,A -85,B 0,C 180,E1 -5007.053,E2 -5007.053} C_VEL
LIN {X 0,Y 516.891,Z 480.914,A -85,B 0,C 180,E1 -5009.796,E2 -5009.796} C_VEL
LIN {X 0,Y 516.929,Z 480.908,A -85,B 0,C 180,E1 -5012.467,E2 -5012.467} C_VEL
LIN {X 0,Y 516.91,Z 480.909,A -85,B 0,C 180,E1 -5015.072,E2 -5015.072} C_VEL
LIN {X 0,Y 516.885,Z 480.913,A -85,B 0,C 180,E1 -5018.462,E2 -5018.462} C_VEL
LIN {X 0,Y 516.902,Z 480.91,A -85,B 0,C 180,E1 -5020.955,E2 -5020.955} C_VEL
LIN {X 0,Y 516.913,Z 480.91,A -85,B 0,C 180,E1 -5023.41,E2 -5023.41} C_VEL
LIN {X 0,Y 516.894,Z 480.913,A -85,B 0,C 180,E1 -5025.834,E2 -5025.834} C_VEL
LIN {X 0,Y 517.002,Z 480.9,A -85,B 0,C 180,E1 -5028.234,E2 -5028.234} C_VEL
LIN {X 0,Y 516.968,Z 480.903,A -85,B 0,C 180,E1 -5031.4,E2 -5031.4} C_VEL
LIN {X 0,Y 517.008,Z 480.898,A -85,B 0,C 180,E1 -5033.757,E2 -5033.757} C_VEL
LIN {X 0,Y 517.084,Z 480.889,A -85,B 0,C 180,E1 -5037.663,E2 -5037.663} C_VEL
LIN {X 0,Y 517.092,Z 480.886,A -85,B 0,C 180,E1 -5040.779,E2 -5040.779} C_VEL
LIN {X 0,Y 517.015,Z 480.897,A -85,B 0,C 180,E1 -5043.117,E2 -5043.117} C_VEL
LIN {X 0,Y 517.01,Z 480.899,A -85,B 0,C 180,E1 -5046.243,E2 -5046.243} C_VEL
LIN {X 0,Y 516.953,Z 480.905,A -85,B 0,C 180,E1 -5049.389,E2 -5049.389} C_VEL
LIN {X 0,Y 516.95,Z 480.906,A -85,B 0,C 180,E1 -5051.808,E2 -5051.808} C_VEL
LIN {X 0,Y 516.942,Z 480.906,A -85,B 0,C 180,E1 -5055.147,E2 -5055.147} C_VEL
LIN {X 0,Y 516.924,Z 480.909,A -85,B 0,C 180,E1 -5058.222,E2 -5058.222} C_VEL
LIN {X 0,Y 516.91,Z 480.911,A -85,B 0,C 180,E1 -5060.702,E2 -5060.702} C_VEL
LIN {X 0,Y 516.909,Z 480.911,A -85,B 0,C 180,E1 -5064.072,E2 -5064.072} C_VEL
LIN {X 0,Y 516.924,Z 480.908,A -85,B 0,C 180,E1 -5066.658,E2 -5066.658} C_VEL
LIN {X 0,Y 516.923,Z 480.909,A -85,B 0,C 180,E1 -5069.527,E2 -5069.527} C_VEL
LIN {X 0,Y 516.899,Z 480.911,A -85,B 0,C 180,E1 -5072.545,E2 -5072.545} C_VEL
LIN {X 0,Y 516.881,Z 480.914,A -85,B 0,C 180,E1 -5075.333,E2 -5075.333} C_VEL
LIN {X 0,Y 516.879,Z 480.916,A -85,B 0,C 180,E1 -5077.943,E2 -5077.943} C_VEL
LIN {X 0,Y 516.883,Z 480.915,A -85,B 0,C 180,E1 -5080.742,E2 -5080.742} C_VEL
LIN {X 0,Y 516.903,Z 480.912,A -85,B 0,C 180,E1 -5082.829,E2 -5082.829} C_VEL
LIN {X 0,Y 516.92,Z 480.909,A -85,B 0,C 180,E1 -5085.01,E2 -5085.01} C_VEL
LIN {X 0,Y 516.921,Z 480.909,A -85,B 0,C 180,E1 -5088.398,E2 -5088.398} C_VEL
LIN {X 0,Y 516.905,Z 480.913,A -85,B 0,C 180,E1 -5091.287,E2 -5091.287} C_VEL
LIN {X 0,Y 516.89,Z 480.913,A -85,B 0,C 180,E1 -5094.222,E2 -5094.222} C_VEL
LIN {X 0,Y 516.931,Z 481.054,A -85,B 0,C 180,E1 -5096.707,E2 -5096.707} C_VEL
LIN {X 0,Y 517.832,Z 486.808,A -85,B 0,C 180,E1 -5098.763,E2 -5098.763} C_VEL
LIN {X 0,Y 517.628,Z 494.031,A -85,B 0,C 180,E1 -5101.185,E2 -5101.185} C_VEL
LIN {X 0,Y 517.365,Z 501.787,A -85,B 0,C 180,E1 -5103.709,E2 -5103.709} C_VEL
LIN {X 0,Y 517.117,Z 511.518,A -85,B 0,C 180,E1 -5106.789,E2 -5106.789} C_VEL
LIN {X 0,Y 516.915,Z 521.093,A -85,B 0,C 180,E1 -5109.739,E2 -5109.739} C_VEL
LIN {X 0,Y 516.735,Z 531.884,A -85,B 0,C 180,E1 -5112.998,E2 -5112.998} C_VEL
LIN {X 0,Y 516.593,Z 541.583,A -85,B 0,C 180,E1 -5115.826,E2 -5115.826} C_VEL
LIN {X 0,Y 516.488,Z 552.56,A -85,B 0,C 180,E1 -5119.018,E2 -5119.018} C_VEL
LIN {X 0,Y 517.569,Z 563.006,A -85,B 0,C 180,E1 -5119.339,E2 -5119.339} C_VEL
LIN {X 0,Y 517.394,Z 574.889,A -85,B 0,C 180,E1 -5119.83,E2 -5119.83} C_VEL
LIN {X 0,Y 517.217,Z 583.646,A -85,B 0,C 180,E1 -5120.32,E2 -5120.32} C_VEL
LIN {X 0,Y 517.069,Z 592.014,A -85,B 0,C 180,E1 -5120.909,E2 -5120.909} C_VEL
LIN {X 0,Y 516.862,Z 599.931,A -85,B 0,C 180,E1 -5121.595,E2 -5121.595} C_VEL
LIN {X 0,Y 516.697,Z 607.337,A -85,B 0,C 180,E1 -5122.38,E2 -5122.38} C_VEL
LIN {X 0,Y 516.525,Z 614.74,A -85,B 0,C 180,E1 -5123.343,E2 -5123.343} C_VEL
LIN {X 0,Y 516.476,Z 620.756,A -85,B 0,C 180,E1 -5124.339,E2 -5124.339} C_VEL
LIN {X 0,Y 516.322,Z 625.396,A -85,B 0,C 180,E1 -5125.316,E2 -5125.316} C_VEL
LIN {X 0,Y 516.367,Z 628.415,A -85,B 0,C 180,E1 -5126.098,E2 -5126.098} C_VEL
LIN {X 0,Y 516.295,Z 630.751,A -85,B 0,C 180,E1 -5126.879,E2 -5126.879} C_VEL
LIN {X 0,Y 516.262,Z 632.509,A -85,B 0,C 180,E1 -5127.66,E2 -5127.66} C_VEL
LIN {X 0,Y 516.191,Z 633.767,A -85,B 0,C 180,E1 -5128.44,E2 -5128.44} C_VEL
LIN {X 0,Y 516.158,Z 634.549,A -85,B 0,C 180,E1 -5129.22,E2 -5129.22} C_VEL
LIN {X 0,Y 516.151,Z 634.845,A -85,B 0,C 180,E1 -5130,E2 -5130} C_VEL
LIN {X 0,Y 516.158,Z 634.548,A -85,B 0,C 180,E1 -5130.781,E2 -5130.781} C_VEL
LIN {X 0,Y 516.191,Z 633.762,A -85,B 0,C 180,E1 -5131.561,E2 -5131.561} C_VEL
LIN {X 0,Y 516.263,Z 632.501,A -85,B 0,C 180,E1 -5132.341,E2 -5132.341} C_VEL
LIN {X 0,Y 516.33,Z 629.578,A -85,B 0,C 180,E1 -5133.512,E2 -5133.512} C_VEL
LIN {X 0,Y 516.376,Z 626.909,A -85,B 0,C 180,E1 -5134.293,E2 -5134.293} C_VEL
LIN {X 0,Y 516.432,Z 621.688,A -85,B 0,C 180,E1 -5135.467,E2 -5135.467} C_VEL
LIN {X 0,Y 516.57,Z 615.867,A -85,B 0,C 180,E1 -5136.478,E2 -5136.478} C_VEL
LIN {X 0,Y 516.659,Z 608.978,A -85,B 0,C 180,E1 -5137.425,E2 -5137.425} C_VEL
LIN {X 0,Y 516.832,Z 600.869,A -85,B 0,C 180,E1 -5138.308,E2 -5138.308} C_VEL
LIN {X 0,Y 517.037,Z 593.13,A -85,B 0,C 180,E1 -5138.994,E2 -5138.994} C_VEL
LIN {X 0,Y 517.177,Z 584.996,A -85,B 0,C 180,E1 -5139.583,E2 -5139.583} C_VEL
LIN {X 0,Y 517.362,Z 576.572,A -85,B 0,C 180,E1 -5140.073,E2 -5140.073} C_VEL
LIN {X 0,Y 517.528,Z 567.975,A -85,B 0,C 180,E1 -5140.465,E2 -5140.465} C_VEL
LIN {X 0,Y 517.37,Z 561.048,A -85,B 0,C 180,E1 -5140.716,E2 -5140.716} C_VEL
LIN {X 0,Y 516.439,Z 552.674,A -85,B 0,C 180,E1 -5140.984,E2 -5140.984} C_VEL
LIN {X 0,Y 516.511,Z 542.156,A -85,B 0,C 180,E1 -5144.178,E2 -5144.178} C_VEL
LIN {X 0,Y 516.608,Z 532.879,A -85,B 0,C 180,E1 -5147.007,E2 -5147.007} C_VEL
LIN {X 0,Y 516.758,Z 525.047,A -85,B 0,C 180,E1 -5149.464,E2 -5149.464} C_VEL
LIN {X 0,Y 516.946,Z 514.641,A -85,B 0,C 180,E1 -5152.797,E2 -5152.797} C_VEL
LIN {X 0,Y 517.101,Z 505.706,A -85,B 0,C 180,E1 -5155.78,E2 -5155.78} C_VEL
LIN {X 0,Y 517.327,Z 498.297,A -85,B 0,C 180,E1 -5158.391,E2 -5158.391} C_VEL
LIN {X 0,Y 517.637,Z 490.889,A -85,B 0,C 180,E1 -5161.201,E2 -5161.201} C_VEL
LIN {X 0,Y 517.79,Z 486.84,A -85,B 0,C 180,E1 -5162.883,E2 -5162.883} C_VEL
LIN {X 0,Y 517.223,Z 482.771,A -85,B 0,C 180,E1 -5164.799,E2 -5164.799} C_VEL
LIN {X 0,Y 516.913,Z 480.912,A -85,B 0,C 180,E1 -5165.777,E2 -5165.777} C_VEL
LIN {X 0,Y 516.89,Z 480.914,A -85,B 0,C 180,E1 -5169.194,E2 -5169.194} C_VEL
LIN {X 0,Y 516.915,Z 480.912,A -85,B 0,C 180,E1 -5171.775,E2 -5171.775} C_VEL
LIN {X 0,Y 516.925,Z 480.911,A -85,B 0,C 180,E1 -5175.01,E2 -5175.01} C_VEL
LIN {X 0,Y 516.919,Z 480.911,A -85,B 0,C 180,E1 -5178.399,E2 -5178.399} C_VEL
LIN {X 0,Y 516.883,Z 480.916,A -85,B 0,C 180,E1 -5181.284,E2 -5181.284} C_VEL
LIN {X 0,Y 516.874,Z 480.916,A -85,B 0,C 180,E1 -5184.22,E2 -5184.22} C_VEL
LIN {X 0,Y 516.862,Z 480.917,A -85,B 0,C 180,E1 -5187.051,E2 -5187.051} C_VEL
LIN {X 0,Y 516.783,Z 480.929,A -85,B 0,C 180,E1 -5187.969,E2 -5187.969} C_VEL
LIN {X 0,Y 516.699,Z 483.927,A -85,B 0,C 180,E1 -5190.682,E2 -5190.682} C_VEL
LIN {X 0,Y 516.599,Z 487.094,A -85,B 0,C 180,E1 -5193.324,E2 -5193.324} C_VEL
LIN {X 0,Y 516.564,Z 490.276,A -85,B 0,C 180,E1 -5195.911,E2 -5195.911} C_VEL
LIN {X 0,Y 516.468,Z 494.546,A -85,B 0,C 180,E1 -5199.28,E2 -5199.28} C_VEL
LIN {X 0,Y 516.376,Z 498.866,A -85,B 0,C 180,E1 -5202.577,E2 -5202.577} C_VEL
LIN {X 0,Y 516.366,Z 503.122,A -85,B 0,C 180,E1 -5205.819,E2 -5205.819} C_VEL
LIN {X 0,Y 516.277,Z 507.643,A -85,B 0,C 180,E1 -5209.162,E2 -5209.162} C_VEL
LIN {X 0,Y 517.552,Z 516.982,A -85,B 0,C 180,E1 -5209.486,E2 -5209.486} C_VEL
LIN {X 0,Y 517.428,Z 526.962,A -85,B 0,C 180,E1 -5209.929,E2 -5209.929} C_VEL
LIN {X 0,Y 517.242,Z 535.482,A -85,B 0,C 180,E1 -5210.419,E2 -5210.419} C_VEL
LIN {X 0,Y 517.098,Z 543.657,A -85,B 0,C 180,E1 -5211.008,E2 -5211.008} C_VEL
LIN {X 0,Y 516.905,Z 551.412,A -85,B 0,C 180,E1 -5211.694,E2 -5211.694} C_VEL
LIN {X 0,Y 516.748,Z 557.814,A -85,B 0,C 180,E1 -5212.38,E2 -5212.38} C_VEL
LIN {X 0,Y 516.626,Z 564.535,A -85,B 0,C 180,E1 -5213.252,E2 -5213.252} C_VEL
LIN {X 0,Y 516.499,Z 571.247,A -85,B 0,C 180,E1 -5214.339,E2 -5214.339} C_VEL
LIN {X 0,Y 516.359,Z 575.898,A -85,B 0,C 180,E1 -5215.316,E2 -5215.316} C_VEL
LIN {X 0,Y 516.39,Z 578.889,A -85,B 0,C 180,E1 -5216.098,E2 -5216.098} C_VEL
LIN {X 0,Y 516.312,Z 581.213,A -85,B 0,C 180,E1 -5216.879,E2 -5216.879} C_VEL
LIN {X 0,Y 516.263,Z 582.987,A -85,B 0,C 180,E1 -5217.659,E2 -5217.659} C_VEL
LIN {X 0,Y 516.192,Z 584.269,A -85,B 0,C 180,E1 -5218.44,E2 -5218.44} C_VEL
LIN {X 0,Y 516.158,Z 585.079,A -85,B 0,C 180,E1 -5219.22,E2 -5219.22} C_VEL
LIN {X 0,Y 516.152,Z 585.383,A -85,B 0,C 180,E1 -5220,E2 -5220} C_VEL
LIN {X 0,Y 516.159,Z 585.112,A -85,B 0,C 180,E1 -5220.78,E2 -5220.78} C_VEL
LIN {X 0,Y 516.191,Z 584.369,A -85,B 0,C 180,E1 -5221.56,E2 -5221.56} C_VEL
LIN {X 0,Y 516.262,Z 583.156,A -85,B 0,C 180,E1 -5222.341,E2 -5222.341} C_VEL
LIN {X 0,Y 516.323,Z 580.309,A -85,B 0,C 180,E1 -5223.512,E2 -5223.512} C_VEL
LIN {X 0,Y 516.392,Z 577.714,A -85,B 0,C 180,E1 -5224.293,E2 -5224.293} C_VEL
LIN {X 0,Y 516.431,Z 572.613,A -85,B 0,C 180,E1 -5225.466,E2 -5225.466} C_VEL
LIN {X 0,Y 516.611,Z 566.674,A -85,B 0,C 180,E1 -5226.513,E2 -5226.513} C_VEL
LIN {X 0,Y 516.688,Z 560.197,A -85,B 0,C 180,E1 -5227.425,E2 -5227.425} C_VEL
LIN {X 0,Y 516.888,Z 552.256,A -85,B 0,C 180,E1 -5228.306,E2 -5228.306} C_VEL
LIN {X 0,Y 517.088,Z 544.681,A -85,B 0,C 180,E1 -5228.992,E2 -5228.992} C_VEL
LIN {X 0,Y 517.249,Z 536.742,A -85,B 0,C 180,E1 -5229.581,E2 -5229.581} C_VEL
LIN {X 0,Y 517.424,Z 528.542,A -85,B 0,C 180,E1 -5230.072,E2 -5230.072} C_VEL
LIN {X 0,Y 517.531,Z 520.24,A -85,B 0,C 180,E1 -5230.465,E2 -5230.465} C_VEL
LIN {X 0,Y 517.248,Z 513.783,A -85,B 0,C 180,E1 -5230.718,E2 -5230.718} C_VEL
LIN {X 0,Y 516.293,Z 507.11,A -85,B 0,C 180,E1 -5230.962,E2 -5230.962} C_VEL
LIN {X 0,Y 516.329,Z 502.251,A -85,B 0,C 180,E1 -5234.182,E2 -5234.182} C_VEL
LIN {X 0,Y 516.364,Z 497.522,A -85,B 0,C 180,E1 -5237.424,E2 -5237.424} C_VEL
LIN {X 0,Y 516.427,Z 493.532,A -85,B 0,C 180,E1 -5240.113,E2 -5240.113} C_VEL
LIN {X 0,Y 516.443,Z 488.99,A -85,B 0,C 180,E1 -5243.244,E2 -5243.244} C_VEL
LIN {X 0,Y 516.512,Z 484.847,A -85,B 0,C 180,E1 -5246.098,E2 -5246.098} C_VEL
LIN {X 0,Y 516.604,Z 483.26,A -85,B 0,C 180,E1 -5247.277,E2 -5247.277} C_VEL
LIN {X 0,Y 516.612,Z 488.612,A -85,B 0,C 180,E1 -5249.464,E2 -5249.464} C_VEL
LIN {X 0,Y 516.624,Z 495.926,A -85,B 0,C 180,E1 -5252.495,E2 -5252.495} C_VEL
LIN {X 0,Y 516.507,Z 502.499,A -85,B 0,C 180,E1 -5255.273,E2 -5255.273} C_VEL
LIN {X 0,Y 516.465,Z 509.576,A -85,B 0,C 180,E1 -5258.288,E2 -5258.288} C_VEL
LIN {X 0,Y 516.4,Z 515.441,A -85,B 0,C 180,E1 -5260.788,E2 -5260.788} C_VEL
LIN {X 0,Y 516.364,Z 522.385,A -85,B 0,C 180,E1 -5263.833,E2 -5263.833} C_VEL
LIN {X 0,Y 516.338,Z 524.809,A -85,B 0,C 180,E1 -5264.906,E2 -5264.906} C_VEL
LIN {X 0,Y 516.341,Z 526.094,A -85,B 0,C 180,E1 -5265.085,E2 -5265.085} C_VEL
LIN {X 0,Y 516.356,Z 529.563,A -85,B 0,C 180,E1 -5265.22,E2 -5265.22} C_VEL
LIN {X 0,Y 515.95,Z 537.876,A -85,B 0,C 180,E1 -5265.488,E2 -5265.488} C_VEL
LIN {X 0,Y 515.18,Z 541.42,A -85,B 0,C 180,E1 -5265.616,E2 -5265.616} C_VEL
LIN {X 0,Y 511.068,Z 550.57,A -85,B 0,C 180,E1 -5265.973,E2 -5265.973} C_VEL
LIN {X 0,Y 510.3,Z 553.766,A -85,B 0,C 180,E1 -5266.169,E2 -5266.169} C_VEL
LIN {X 0,Y 510.035,Z 564.044,A -85,B 0,C 180,E1 -5266.912,E2 -5266.912} C_VEL
LIN {X 0,Y 509.805,Z 572.393,A -85,B 0,C 180,E1 -5267.678,E2 -5267.678} C_VEL
LIN {X 0,Y 509.615,Z 580.092,A -85,B 0,C 180,E1 -5268.55,E2 -5268.55} C_VEL
LIN {X 0,Y 509.444,Z 587.305,A -85,B 0,C 180,E1 -5269.58,E2 -5269.58} C_VEL
LIN {X 0,Y 509.326,Z 592.907,A -85,B 0,C 180,E1 -5270.599,E2 -5270.599} C_VEL
LIN {X 0,Y 509.262,Z 597.257,A -85,B 0,C 180,E1 -5271.609,E2 -5271.609} C_VEL
LIN {X 0,Y 509.213,Z 600.549,A -85,B 0,C 180,E1 -5272.607,E2 -5272.607} C_VEL
LIN {X 0,Y 509.124,Z 602.904,A -85,B 0,C 180,E1 -5273.588,E2 -5273.588} C_VEL
LIN {X 0,Y 509.091,Z 604.429,A -85,B 0,C 180,E1 -5274.562,E2 -5274.562} C_VEL
LIN {X 0,Y 509.078,Z 605.339,A -85,B 0,C 180,E1 -5275.927,E2 -5275.927} C_VEL
LIN {X 0,Y 509.092,Z 604.546,A -85,B 0,C 180,E1 -5277.425,E2 -5277.425} C_VEL
LIN {X 0,Y 509.156,Z 602.168,A -85,B 0,C 180,E1 -5278.848,E2 -5278.848} C_VEL
LIN {X 0,Y 509.23,Z 598.264,A -85,B 0,C 180,E1 -5280.208,E2 -5280.208} C_VEL
LIN {X 0,Y 509.322,Z 593.568,A -85,B 0,C 180,E1 -5281.347,E2 -5281.347} C_VEL
LIN {X 0,Y 509.475,Z 587.496,A -85,B 0,C 180,E1 -5282.476,E2 -5282.476} C_VEL
LIN {X 0,Y 509.635,Z 579.976,A -85,B 0,C 180,E1 -5283.551,E2 -5283.551} C_VEL
LIN {X 0,Y 509.826,Z 572.761,A -85,B 0,C 180,E1 -5284.373,E2 -5284.373} C_VEL
LIN {X 0,Y 510.044,Z 564.935,A -85,B 0,C 180,E1 -5285.1,E2 -5285.1} C_VEL
LIN {X 0,Y 510.258,Z 555.44,A -85,B 0,C 180,E1 -5285.81,E2 -5285.81} C_VEL
LIN {X 0,Y 510.473,Z 544.779,A -85,B 0,C 180,E1 -5286.414,E2 -5286.414} C_VEL
LIN {X 0,Y 510.505,Z 535.042,A -85,B 0,C 180,E1 -5286.818,E2 -5286.818} C_VEL
LIN {X 0,Y 509.206,Z 525.681,A -85,B 0,C 180,E1 -5287.132,E2 -5287.132} C_VEL
LIN {X 0,Y 509.263,Z 519.892,A -85,B 0,C 180,E1 -5289.817,E2 -5289.817} C_VEL
LIN {X 0,Y 509.36,Z 514.564,A -85,B 0,C 180,E1 -5292.329,E2 -5292.329} C_VEL
LIN {X 0,Y 509.44,Z 507.499,A -85,B 0,C 180,E1 -5295.622,E2 -5295.622} C_VEL
LIN {X 0,Y 509.515,Z 500.417,A -85,B 0,C 180,E1 -5298.865,E2 -5298.865} C_VEL
LIN {X 0,Y 509.535,Z 493.429,A -85,B 0,C 180,E1 -5302.072,E2 -5302.072} C_VEL
LIN {X 0,Y 509.569,Z 488.177,A -85,B 0,C 180,E1 -5304.459,E2 -5304.459} C_VEL
LIN {X 0,Y 509.503,Z 482.901,A -85,B 0,C 180,E1 -5306.837,E2 -5306.837} C_VEL
LIN {X 0,Y 509.568,Z 481.827,A -85,B 0,C 180,E1 -5307.431,E2 -5307.431} C_VEL
LIN {X 0,Y 510.04,Z 481.767,A -85,B 0,C 180,E1 -5309.21,E2 -5309.21} C_VEL
LIN {X 0,Y 509.934,Z 481.779,A -85,B 0,C 180,E1 -5311.579,E2 -5311.579} C_VEL
LIN {X 0,Y 509.956,Z 481.776,A -85,B 0,C 180,E1 -5313.16,E2 -5313.16} C_VEL
LIN {X 0,Y 509.983,Z 481.775,A -85,B 0,C 180,E1 -5316.329,E2 -5316.329} C_VEL
LIN {X 0,Y 509.914,Z 481.784,A -85,B 0,C 180,E1 -5318.72,E2 -5318.72} C_VEL
LIN {X 0,Y 509.906,Z 481.783,A -85,B 0,C 180,E1 -5321.931,E2 -5321.931} C_VEL
LIN {X 0,Y 509.895,Z 481.782,A -85,B 0,C 180,E1 -5325.241,E2 -5325.241} C_VEL
LIN {X 0,Y 509.89,Z 481.785,A -85,B 0,C 180,E1 -5328.001,E2 -5328.001} C_VEL
LIN {X 0,Y 509.851,Z 481.788,A -85,B 0,C 180,E1 -5331.001,E2 -5331.001} C_VEL
LIN {X 0,Y 509.837,Z 481.791,A -85,B 0,C 180,E1 -5333.563,E2 -5333.563} C_VEL
LIN {X 0,Y 509.914,Z 481.784,A -85,B 0,C 180,E1 -5336.379,E2 -5336.379} C_VEL
LIN {X 0,Y 509.882,Z 481.787,A -85,B 0,C 180,E1 -5338.843,E2 -5338.843} C_VEL
LIN {X 0,Y 509.827,Z 481.793,A -85,B 0,C 180,E1 -5341.589,E2 -5341.589} C_VEL
LIN {X 0,Y 509.854,Z 481.79,A -85,B 0,C 180,E1 -5344.413,E2 -5344.413} C_VEL
LIN {X 0,Y 509.819,Z 481.795,A -85,B 0,C 180,E1 -5347.34,E2 -5347.34} C_VEL
LIN {X 0,Y 509.837,Z 481.792,A -85,B 0,C 180,E1 -5350.382,E2 -5350.382} C_VEL
LIN {X 0,Y 509.838,Z 481.792,A -85,B 0,C 180,E1 -5353.064,E2 -5353.064} C_VEL
LIN {X 0,Y 509.829,Z 481.793,A -85,B 0,C 180,E1 -5355.792,E2 -5355.792} C_VEL
LIN {X 0,Y 509.865,Z 481.788,A -85,B 0,C 180,E1 -5358.575,E2 -5358.575} C_VEL
LIN {X 0,Y 509.854,Z 481.79,A -85,B 0,C 180,E1 -5361.785,E2 -5361.785} C_VEL
LIN {X 0,Y 509.828,Z 481.794,A -85,B 0,C 180,E1 -5364.622,E2 -5364.622} C_VEL
LIN {X 0,Y 509.864,Z 481.789,A -85,B 0,C 180,E1 -5367.481,E2 -5367.481} C_VEL
LIN {X 0,Y 509.856,Z 481.789,A -85,B 0,C 180,E1 -5370.273,E2 -5370.273} C_VEL
LIN {X 0,Y 509.886,Z 481.786,A -85,B 0,C 180,E1 -5372.944,E2 -5372.944} C_VEL
LIN {X 0,Y 509.869,Z 481.789,A -85,B 0,C 180,E1 -5375.574,E2 -5375.574} C_VEL
LIN {X 0,Y 509.821,Z 481.794,A -85,B 0,C 180,E1 -5378.149,E2 -5378.149} C_VEL
LIN {X 0,Y 509.862,Z 481.787,A -85,B 0,C 180,E1 -5380.681,E2 -5380.681} C_VEL
LIN {X 0,Y 509.883,Z 481.785,A -85,B 0,C 180,E1 -5383.175,E2 -5383.175} C_VEL
LIN {X 0,Y 509.863,Z 481.788,A -85,B 0,C 180,E1 -5385.634,E2 -5385.634} C_VEL
LIN {X 0,Y 509.92,Z 481.78,A -85,B 0,C 180,E1 -5388.875,E2 -5388.875} C_VEL
LIN {X 0,Y 509.95,Z 481.779,A -85,B 0,C 180,E1 -5392.078,E2 -5392.078} C_VEL
LIN {X 0,Y 509.98,Z 481.774,A -85,B 0,C 180,E1 -5394.464,E2 -5394.464} C_VEL
LIN {X 0,Y 510.055,Z 481.765,A -85,B 0,C 180,E1 -5397.631,E2 -5397.631} C_VEL
LIN {X 0,Y 510.062,Z 481.762,A -85,B 0,C 180,E1 -5400.789,E2 -5400.789} C_VEL
LIN {X 0,Y 509.957,Z 481.776,A -85,B 0,C 180,E1 -5403.16,E2 -5403.16} C_VEL
LIN {X 0,Y 509.978,Z 481.774,A -85,B 0,C 180,E1 -5406.33,E2 -5406.33} C_VEL
LIN {X 0,Y 509.915,Z 481.782,A -85,B 0,C 180,E1 -5408.72,E2 -5408.72} C_VEL
LIN {X 0,Y 509.902,Z 481.785,A -85,B 0,C 180,E1 -5411.932,E2 -5411.932} C_VEL
LIN {X 0,Y 509.891,Z 481.784,A -85,B 0,C 180,E1 -5415.242,E2 -5415.242} C_VEL
LIN {X 0,Y 509.886,Z 481.787,A -85,B 0,C 180,E1 -5418.001,E2 -5418.001} C_VEL
LIN {X 0,Y 509.848,Z 481.789,A -85,B 0,C 180,E1 -5421.002,E2 -5421.002} C_VEL
LIN {X 0,Y 509.835,Z 481.792,A -85,B 0,C 180,E1 -5423.563,E2 -5423.563} C_VEL
LIN {X 0,Y 509.909,Z 481.783,A -85,B 0,C 180,E1 -5426.379,E2 -5426.379} C_VEL
LIN {X 0,Y 509.883,Z 481.787,A -85,B 0,C 180,E1 -5428.844,E2 -5428.844} C_VEL
LIN {X 0,Y 509.825,Z 481.793,A -85,B 0,C 180,E1 -5431.59,E2 -5431.59} C_VEL
LIN {X 0,Y 509.852,Z 481.79,A -85,B 0,C 180,E1 -5434.413,E2 -5434.413} C_VEL
LIN {X 0,Y 509.817,Z 481.794,A -85,B 0,C 180,E1 -5437.341,E2 -5437.341} C_VEL
LIN {X 0,Y 509.836,Z 481.792,A -85,B 0,C 180,E1 -5440.382,E2 -5440.382} C_VEL
LIN {X 0,Y 509.838,Z 481.793,A -85,B 0,C 180,E1 -5443.065,E2 -5443.065} C_VEL
LIN {X 0,Y 509.828,Z 481.792,A -85,B 0,C 180,E1 -5445.793,E2 -5445.793} C_VEL
LIN {X 0,Y 509.864,Z 481.788,A -85,B 0,C 180,E1 -5448.576,E2 -5448.576} C_VEL
LIN {X 0,Y 509.857,Z 481.789,A -85,B 0,C 180,E1 -5451.663,E2 -5451.663} C_VEL
LIN {X 0,Y 509.845,Z 481.793,A -85,B 0,C 180,E1 -5454.624,E2 -5454.624} C_VEL
LIN {X 0,Y 509.887,Z 481.838,A -85,B 0,C 180,E1 -5456.483,E2 -5456.483} C_VEL
LIN {X 0,Y 510.814,Z 487.497,A -85,B 0,C 180,E1 -5458.542,E2 -5458.542} C_VEL
LIN {X 0,Y 510.655,Z 493.965,A -85,B 0,C 180,E1 -5460.753,E2 -5460.753} C_VEL
LIN {X 0,Y 510.391,Z 502.292,A -85,B 0,C 180,E1 -5463.513,E2 -5463.513} C_VEL
LIN {X 0,Y 510.099,Z 511.394,A -85,B 0,C 180,E1 -5466.45,E2 -5466.45} C_VEL
LIN {X 0,Y 509.938,Z 519.51,A -85,B 0,C 180,E1 -5469.003,E2 -5469.003} C_VEL
LIN {X 0,Y 509.708,Z 529.451,A -85,B 0,C 180,E1 -5472.062,E2 -5472.062} C_VEL
LIN {X 0,Y 509.539,Z 540.12,A -85,B 0,C 180,E1 -5475.263,E2 -5475.263} C_VEL
LIN {X 0,Y 509.459,Z 550.565,A -85,B 0,C 180,E1 -5478.363,E2 -5478.363} C_VEL
LIN {X 0,Y 509.407,Z 552.49,A -85,B 0,C 180,E1 -5478.889,E2 -5478.889} C_VEL
LIN {X 0,Y 510.585,Z 564.062,A -85,B 0,C 180,E1 -5479.241,E2 -5479.241} C_VEL
LIN {X 0,Y 510.378,Z 574.455,A -85,B 0,C 180,E1 -5479.688,E2 -5479.688} C_VEL
LIN {X 0,Y 510.217,Z 583.224,A -85,B 0,C 180,E1 -5480.186,E2 -5480.186} C_VEL
LIN {X 0,Y 510.051,Z 591.603,A -85,B 0,C 180,E1 -5480.783,E2 -5480.783} C_VEL
LIN {X 0,Y 509.816,Z 599.531,A -85,B 0,C 180,E1 -5481.478,E2 -5481.478} C_VEL
LIN {X 0,Y 509.625,Z 606.947,A -85,B 0,C 180,E1 -5482.273,E2 -5482.273} C_VEL
LIN {X 0,Y 509.441,Z 615.053,A -85,B 0,C 180,E1 -5483.352,E2 -5483.352} C_VEL
LIN {X 0,Y 509.355,Z 621.362,A -85,B 0,C 180,E1 -5484.458,E2 -5484.458} C_VEL
LIN {X 0,Y 509.267,Z 626.578,A -85,B 0,C 180,E1 -5485.647,E2 -5485.647} C_VEL
LIN {X 0,Y 509.246,Z 629.248,A -85,B 0,C 180,E1 -5486.44,E2 -5486.44} C_VEL
LIN {X 0,Y 509.191,Z 632.172,A -85,B 0,C 180,E1 -5487.627,E2 -5487.627} C_VEL
LIN {X 0,Y 509.111,Z 633.431,A -85,B 0,C 180,E1 -5488.418,E2 -5488.418} C_VEL
LIN {X 0,Y 509.071,Z 634.214,A -85,B 0,C 180,E1 -5489.209,E2 -5489.209} C_VEL
LIN {X 0,Y 509.063,Z 634.506,A -85,B 0,C 180,E1 -5490,E2 -5490} C_VEL
LIN {X 0,Y 509.071,Z 634.208,A -85,B 0,C 180,E1 -5490.791,E2 -5490.791} C_VEL
LIN {X 0,Y 509.111,Z 633.418,A -85,B 0,C 180,E1 -5491.582,E2 -5491.582} C_VEL
LIN {X 0,Y 509.192,Z 632.148,A -85,B 0,C 180,E1 -5492.374,E2 -5492.374} C_VEL
LIN {X 0,Y 509.25,Z 629.213,A -85,B 0,C 180,E1 -5493.561,E2 -5493.561} C_VEL
LIN {X 0,Y 509.267,Z 626.529,A -85,B 0,C 180,E1 -5494.353,E2 -5494.353} C_VEL
LIN {X 0,Y 509.355,Z 621.293,A -85,B 0,C 180,E1 -5495.543,E2 -5495.543} C_VEL
LIN {X 0,Y 509.518,Z 614.445,A -85,B 0,C 180,E1 -5496.722,E2 -5496.722} C_VEL
LIN {X 0,Y 509.626,Z 606.809,A -85,B 0,C 180,E1 -5497.728,E2 -5497.728} C_VEL
LIN {X 0,Y 509.817,Z 599.36,A -85,B 0,C 180,E1 -5498.523,E2 -5498.523} C_VEL
LIN {X 0,Y 510.043,Z 591.385,A -85,B 0,C 180,E1 -5499.218,E2 -5499.218} C_VEL
LIN {X 0,Y 510.247,Z 581.456,A -85,B 0,C 180,E1 -5499.914,E2 -5499.914} C_VEL
LIN {X 0,Y 510.47,Z 569.805,A -85,B 0,C 180,E1 -5500.511,E2 -5500.511} C_VEL
LIN {X 0,Y 510.422,Z 562.088,A -85,B 0,C 180,E1 -5500.813,E2 -5500.813} C_VEL
LIN {X 0,Y 509.343,Z 552.351,A -85,B 0,C 180,E1 -5501.113,E2 -5501.113} C_VEL
LIN {X 0,Y 509.431,Z 541.794,A -85,B 0,C 180,E1 -5504.379,E2 -5504.379} C_VEL
LIN {X 0,Y 509.553,Z 532.55,A -85,B 0,C 180,E1 -5507.25,E2 -5507.25} C_VEL
LIN {X 0,Y 509.675,Z 524.758,A -85,B 0,C 180,E1 -5509.745,E2 -5509.745} C_VEL
LIN {X 0,Y 509.908,Z 514.381,A -85,B 0,C 180,E1 -5513.13,E2 -5513.13} C_VEL
LIN {X 0,Y 510.079,Z 505.562,A -85,B 0,C 180,E1 -5516.162,E2 -5516.162} C_VEL
LIN {X 0,Y 510.375,Z 498.259,A -85,B 0,C 180,E1 -5518.814,E2 -5518.814} C_VEL
LIN {X 0,Y 510.792,Z 490.256,A -85,B 0,C 180,E1 -5521.987,E2 -5521.987} C_VEL
LIN {X 0,Y 510.751,Z 487.085,A -85,B 0,C 180,E1 -5523.395,E2 -5523.395} C_VEL
LIN {X 0,Y 509.855,Z 481.791,A -85,B 0,C 180,E1 -5526.146,E2 -5526.146} C_VEL
LIN {X 0,Y 509.85,Z 481.791,A -85,B 0,C 180,E1 -5529.353,E2 -5529.353} C_VEL
LIN {X 0,Y 509.836,Z 481.791,A -85,B 0,C 180,E1 -5532.49,E2 -5532.49} C_VEL
LIN {X 0,Y 509.86,Z 481.789,A -85,B 0,C 180,E1 -5535.332,E2 -5535.332} C_VEL
LIN {X 0,Y 509.86,Z 481.79,A -85,B 0,C 180,E1 -5538.575,E2 -5538.575} C_VEL
LIN {X 0,Y 509.854,Z 481.79,A -85,B 0,C 180,E1 -5541.787,E2 -5541.787} C_VEL
LIN {X 0,Y 509.833,Z 481.794,A -85,B 0,C 180,E1 -5544.622,E2 -5544.622} C_VEL
LIN {X 0,Y 509.82,Z 481.796,A -85,B 0,C 180,E1 -5547.478,E2 -5547.478} C_VEL
LIN {X 0,Y 509.759,Z 482.653,A -85,B 0,C 180,E1 -5548.737,E2 -5548.737} C_VEL
LIN {X 0,Y 509.636,Z 485.383,A -85,B 0,C 180,E1 -5551.141,E2 -5551.141} C_VEL
LIN {X 0,Y 509.555,Z 488.537,A -85,B 0,C 180,E1 -5553.81,E2 -5553.81} C_VEL
LIN {X 0,Y 509.446,Z 491.706,A -85,B 0,C 180,E1 -5556.418,E2 -5556.418} C_VEL
LIN {X 0,Y 509.422,Z 495.97,A -85,B 0,C 180,E1 -5559.824,E2 -5559.824} C_VEL
LIN {X 0,Y 509.283,Z 500.276,A -85,B 0,C 180,E1 -5563.154,E2 -5563.154} C_VEL
LIN {X 0,Y 509.309,Z 503.486,A -85,B 0,C 180,E1 -5565.618,E2 -5565.618} C_VEL
LIN {X 0,Y 509.223,Z 508.046,A -85,B 0,C 180,E1 -5569.01,E2 -5569.01} C_VEL
LIN {X 0,Y 510.53,Z 517.191,A -85,B 0,C 180,E1 -5569.34,E2 -5569.34} C_VEL
LIN {X 0,Y 510.453,Z 527.183,A -85,B 0,C 180,E1 -5569.79,E2 -5569.79} C_VEL
LIN {X 0,Y 510.259,Z 535.719,A -85,B 0,C 180,E1 -5570.286,E2 -5570.286} C_VEL
LIN {X 0,Y 510.098,Z 543.91,A -85,B 0,C 180,E1 -5570.883,E2 -5570.883} C_VEL
LIN {X 0,Y 509.905,Z 551.68,A -85,B 0,C 180,E1 -5571.579,E2 -5571.579} C_VEL
LIN {X 0,Y 509.711,Z 558.098,A -85,B 0,C 180,E1 -5572.274,E2 -5572.274} C_VEL
LIN {X 0,Y 509.607,Z 563.998,A -85,B 0,C 180,E1 -5573.04,E2 -5573.04} C_VEL
LIN {X 0,Y 509.541,Z 569.267,A -85,B 0,C 180,E1 -5573.864,E2 -5573.864} C_VEL
LIN {X 0,Y 509.284,Z 574.441,A -85,B 0,C 180,E1 -5574.854,E2 -5574.854} C_VEL
LIN {X 0,Y 509.322,Z 579.223,A -85,B 0,C 180,E1 -5576.044,E2 -5576.044} C_VEL
LIN {X 0,Y 509.228,Z 581.551,A -85,B 0,C 180,E1 -5576.835,E2 -5576.835} C_VEL
LIN {X 0,Y 509.192,Z 583.329,A -85,B 0,C 180,E1 -5577.627,E2 -5577.627} C_VEL
LIN {X 0,Y 509.113,Z 584.613,A -85,B 0,C 180,E1 -5578.418,E2 -5578.418} C_VEL
LIN {X 0,Y 509.071,Z 585.423,A -85,B 0,C 180,E1 -5579.209,E2 -5579.209} C_VEL
LIN {X 0,Y 509.063,Z 585.724,A -85,B 0,C 180,E1 -5580,E2 -5580} C_VEL
LIN {X 0,Y 509.073,Z 585.449,A -85,B 0,C 180,E1 -5580.791,E2 -5580.791} C_VEL
LIN {X 0,Y 509.112,Z 584.703,A -85,B 0,C 180,E1 -5581.582,E2 -5581.582} C_VEL
LIN {X 0,Y 509.191,Z 583.481,A -85,B 0,C 180,E1 -5582.373,E2 -5582.373} C_VEL
LIN {X 0,Y 509.245,Z 580.624,A -85,B 0,C 180,E1 -5583.561,E2 -5583.561} C_VEL
LIN {X 0,Y 509.317,Z 578.015,A -85,B 0,C 180,E1 -5584.353,E2 -5584.353} C_VEL
LIN {X 0,Y 509.382,Z 572.897,A -85,B 0,C 180,E1 -5585.542,E2 -5585.542} C_VEL
LIN {X 0,Y 509.569,Z 567.549,A -85,B 0,C 180,E1 -5586.503,E2 -5586.503} C_VEL
LIN {X 0,Y 509.666,Z 560.434,A -85,B 0,C 180,E1 -5587.527,E2 -5587.527} C_VEL
LIN {X 0,Y 509.883,Z 552.467,A -85,B 0,C 180,E1 -5588.421,E2 -5588.421} C_VEL
LIN {X 0,Y 510.094,Z 544.871,A -85,B 0,C 180,E1 -5589.117,E2 -5589.117} C_VEL
LIN {X 0,Y 510.267,Z 536.908,A -85,B 0,C 180,E1 -5589.714,E2 -5589.714} C_VEL
LIN {X 0,Y 510.451,Z 528.682,A -85,B 0,C 180,E1 -5590.211,E2 -5590.211} C_VEL
LIN {X 0,Y 510.575,Z 520.35,A -85,B 0,C 180,E1 -5590.609,E2 -5590.609} C_VEL
LIN {X 0,Y 510.165,Z 513.857,A -85,B 0,C 180,E1 -5590.869,E2 -5590.869} C_VEL
LIN {X 0,Y 509.247,Z 507.447,A -85,B 0,C 180,E1 -5591.09,E2 -5591.09} C_VEL
LIN {X 0,Y 509.21,Z 503.755,A -85,B 0,C 180,E1 -5593.57,E2 -5593.57} C_VEL
LIN {X 0,Y 509.245,Z 500.127,A -85,B 0,C 180,E1 -5596.023,E2 -5596.023} C_VEL
LIN {X 0,Y 509.297,Z 496.463,A -85,B 0,C 180,E1 -5598.505,E2 -5598.505} C_VEL
LIN {X 0,Y 509.302,Z 492.79,A -85,B 0,C 180,E1 -5601.025,E2 -5601.025} C_VEL
LIN {X 0,Y 509.36,Z 489.123,A -85,B 0,C 180,E1 -5603.587,E2 -5603.587} C_VEL
LIN {X 0,Y 509.463,Z 485.279,A -85,B 0,C 180,E1 -5606.275,E2 -5606.275} C_VEL
LIN {X 0,Y 509.549,Z 484.009,A -85,B 0,C 180,E1 -5607.297,E2 -5607.297} C_VEL
LIN {X 0,Y 509.522,Z 490.092,A -85,B 0,C 180,E1 -5609.773,E2 -5609.773} C_VEL
LIN {X 0,Y 509.571,Z 497.089,A -85,B 0,C 180,E1 -5612.721,E2 -5612.721} C_VEL
LIN {X 0,Y 509.443,Z 503.701,A -85,B 0,C 180,E1 -5615.518,E2 -5615.518} C_VEL
LIN {X 0,Y 509.409,Z 510.347,A -85,B 0,C 180,E1 -5618.377,E2 -5618.377} C_VEL
LIN {X 0,Y 509.322,Z 515.572,A -85,B 0,C 180,E1 -5620.629,E2 -5620.629} C_VEL
LIN {X 0,Y 509.295,Z 522.428,A -85,B 0,C 180,E1 -5623.628,E2 -5623.628} C_VEL
LIN {X 0,Y 509.282,Z 525.453,A -85,B 0,C 180,E1 -5624.95,E2 -5624.95} C_VEL
LIN {X 0,Y 510.636,Z 536.586,A -85,B 0,C 180,E1 -5625.326,E2 -5625.326} C_VEL
LIN {X 0,Y 510.444,Z 548.411,A -85,B 0,C 180,E1 -5625.864,E2 -5625.864} C_VEL
LIN {X 0,Y 510.3,Z 553.766,A -85,B 0,C 180,E1 -5626.169,E2 -5626.169} C_VEL
LIN {X 0,Y 509.59,Z 558.875,A -85,B 0,C 180,E1 -5626.493,E2 -5626.493} C_VEL
LIN {X 0,Y 506.58,Z 566.821,A -85,B 0,C 180,E1 -5627.069,E2 -5627.069} C_VEL
LIN {X 0,Y 503.485,Z 574.203,A -85,B 0,C 180,E1 -5627.741,E2 -5627.741} C_VEL
LIN {X 0,Y 502.652,Z 578.33,A -85,B 0,C 180,E1 -5628.21,E2 -5628.21} C_VEL
LIN {X 0,Y 502.446,Z 584.632,A -85,B 0,C 180,E1 -5629.054,E2 -5629.054} C_VEL
LIN {X 0,Y 502.356,Z 590.066,A -85,B 0,C 180,E1 -5629.943,E2 -5629.943} C_VEL
LIN {X 0,Y 502.207,Z 595.13,A -85,B 0,C 180,E1 -5630.969,E2 -5630.969} C_VEL
LIN {X 0,Y 502.14,Z 599.04,A -85,B 0,C 180,E1 -5631.987,E2 -5631.987} C_VEL
LIN {X 0,Y 502.079,Z 601.922,A -85,B 0,C 180,E1 -5632.993,E2 -5632.993} C_VEL
LIN {X 0,Y 502.006,Z 604.32,A -85,B 0,C 180,E1 -5634.291,E2 -5634.291} C_VEL
LIN {X 0,Y 502.006,Z 605.105,A -85,B 0,C 180,E1 -5634.97,E2 -5634.97} C_VEL
LIN {X 0,Y 502.003,Z 605.535,A -85,B 0,C 180,E1 -5635.944,E2 -5635.944} C_VEL
LIN {X 0,Y 501.972,Z 605.077,A -85,B 0,C 180,E1 -5637.145,E2 -5637.145} C_VEL
LIN {X 0,Y 502.007,Z 604.239,A -85,B 0,C 180,E1 -5637.859,E2 -5637.859} C_VEL
LIN {X 0,Y 502.111,Z 601.422,A -85,B 0,C 180,E1 -5639.277,E2 -5639.277} C_VEL
LIN {X 0,Y 502.139,Z 598.674,A -85,B 0,C 180,E1 -5640.2,E2 -5640.2} C_VEL
LIN {X 0,Y 502.241,Z 594,A -85,B 0,C 180,E1 -5641.362,E2 -5641.362} C_VEL
LIN {X 0,Y 502.329,Z 589.921,A -85,B 0,C 180,E1 -5642.169,E2 -5642.169} C_VEL
LIN {X 0,Y 502.471,Z 585.104,A -85,B 0,C 180,E1 -5642.962,E2 -5642.962} C_VEL
LIN {X 0,Y 502.601,Z 578.434,A -85,B 0,C 180,E1 -5643.866,E2 -5643.866} C_VEL
LIN {X 0,Y 502.846,Z 570.201,A -85,B 0,C 180,E1 -5644.768,E2 -5644.768} C_VEL
LIN {X 0,Y 503.142,Z 561.114,A -85,B 0,C 180,E1 -5645.555,E2 -5645.555} C_VEL
LIN {X 0,Y 503.28,Z 553.047,A -85,B 0,C 180,E1 -5646.111,E2 -5646.111} C_VEL
LIN {X 0,Y 503.518,Z 543.689,A -85,B 0,C 180,E1 -5646.614,E2 -5646.614} C_VEL
LIN {X 0,Y 503.488,Z 535.258,A -85,B 0,C 180,E1 -5646.966,E2 -5646.966} C_VEL
LIN {X 0,Y 502.141,Z 525.852,A -85,B 0,C 180,E1 -5647.294,E2 -5647.294} C_VEL
LIN {X 0,Y 502.209,Z 519.285,A -85,B 0,C 180,E1 -5650.375,E2 -5650.375} C_VEL
LIN {X 0,Y 502.256,Z 513.854,A -85,B 0,C 180,E1 -5652.911,E2 -5652.911} C_VEL
LIN {X 0,Y 502.342,Z 508.552,A -85,B 0,C 180,E1 -5655.414,E2 -5655.414} C_VEL
LIN {X 0,Y 502.448,Z 501.421,A -85,B 0,C 180,E1 -5658.707,E2 -5658.707} C_VEL
LIN {X 0,Y 502.464,Z 494.344,A -85,B 0,C 180,E1 -5661.959,E2 -5661.959} C_VEL
LIN {X 0,Y 502.501,Z 489.062,A -85,B 0,C 180,E1 -5664.381,E2 -5664.381} C_VEL
LIN {X 0,Y 502.445,Z 483.75,A -85,B 0,C 180,E1 -5666.792,E2 -5666.792} C_VEL
LIN {X 0,Y 502.48,Z 482.709,A -85,B 0,C 180,E1 -5667.294,E2 -5667.294} C_VEL
LIN {X 0,Y 502.989,Z 482.645,A -85,B 0,C 180,E1 -5669.199,E2 -5669.199} C_VEL
LIN {X 0,Y 503.037,Z 482.638,A -85,B 0,C 180,E1 -5670.8,E2 -5670.8} C_VEL
LIN {X 0,Y 502.899,Z 482.655,A -85,B 0,C 180,E1 -5673.204,E2 -5673.204} C_VEL
LIN {X 0,Y 502.932,Z 482.654,A -85,B 0,C 180,E1 -5676.418,E2 -5676.418} C_VEL
LIN {X 0,Y 502.872,Z 482.66,A -85,B 0,C 180,E1 -5678.843,E2 -5678.843} C_VEL
LIN {X 0,Y 502.848,Z 482.663,A -85,B 0,C 180,E1 -5682.101,E2 -5682.101} C_VEL
LIN {X 0,Y 502.85,Z 482.66,A -85,B 0,C 180,E1 -5685.399,E2 -5685.399} C_VEL
LIN {X 0,Y 502.847,Z 482.663,A -85,B 0,C 180,E1 -5688.122,E2 -5688.122} C_VEL
LIN {X 0,Y 502.829,Z 482.667,A -85,B 0,C 180,E1 -5690.536,E2 -5690.536} C_VEL
LIN {X 0,Y 502.798,Z 482.669,A -85,B 0,C 180,E1 -5693.04,E2 -5693.04} C_VEL
LIN {X 0,Y 502.842,Z 482.663,A -85,B 0,C 180,E1 -5695.675,E2 -5695.675} C_VEL
LIN {X 0,Y 502.842,Z 482.663,A -85,B 0,C 180,E1 -5698.372,E2 -5698.372} C_VEL
LIN {X 0,Y 502.797,Z 482.669,A -85,B 0,C 180,E1 -5701.499,E2 -5701.499} C_VEL
LIN {X 0,Y 502.806,Z 482.668,A -85,B 0,C 180,E1 -5704.444,E2 -5704.444} C_VEL
LIN {X 0,Y 502.781,Z 482.671,A -85,B 0,C 180,E1 -5707.178,E2 -5707.178} C_VEL
LIN {X 0,Y 502.787,Z 482.67,A -85,B 0,C 180,E1 -5710.015,E2 -5710.015} C_VEL
LIN {X 0,Y 502.801,Z 482.668,A -85,B 0,C 180,E1 -5712.199,E2 -5712.199} C_VEL
LIN {X 0,Y 502.799,Z 482.669,A -85,B 0,C 180,E1 -5715.468,E2 -5715.468} C_VEL
LIN {X 0,Y 502.834,Z 482.666,A -85,B 0,C 180,E1 -5717.865,E2 -5717.865} C_VEL
LIN {X 0,Y 502.81,Z 482.666,A -85,B 0,C 180,E1 -5721.025,E2 -5721.025} C_VEL
LIN {X 0,Y 502.773,Z 482.672,A -85,B 0,C 180,E1 -5724.169,E2 -5724.169} C_VEL
LIN {X 0,Y 502.831,Z 482.664,A -85,B 0,C 180,E1 -5726.993,E2 -5726.993} C_VEL
LIN {X 0,Y 502.813,Z 482.667,A -85,B 0,C 180,E1 -5730.065,E2 -5730.065} C_VEL
LIN {X 0,Y 502.834,Z 482.663,A -85,B 0,C 180,E1 -5732.533,E2 -5732.533} C_VEL
LIN {X 0,Y 502.827,Z 482.664,A -85,B 0,C 180,E1 -5735.298,E2 -5735.298} C_VEL
LIN {X 0,Y 502.783,Z 482.672,A -85,B 0,C 180,E1 -5737.827,E2 -5737.827} C_VEL
LIN {X 0,Y 502.824,Z 482.665,A -85,B 0,C 180,E1 -5740.4,E2 -5740.4} C_VEL
LIN {X 0,Y 502.832,Z 482.664,A -85,B 0,C 180,E1 -5742.932,E2 -5742.932} C_VEL
LIN {X 0,Y 502.843,Z 482.663,A -85,B 0,C 180,E1 -5745.429,E2 -5745.429} C_VEL
LIN {X 0,Y 502.89,Z 482.656,A -85,B 0,C 180,E1 -5748.717,E2 -5748.717} C_VEL
LIN {X 0,Y 502.9,Z 482.658,A -85,B 0,C 180,E1 -5751.967,E2 -5751.967} C_VEL
LIN {X 0,Y 502.936,Z 482.652,A -85,B 0,C 180,E1 -5754.386,E2 -5754.386} C_VEL
LIN {X 0,Y 503.025,Z 482.64,A -85,B 0,C 180,E1 -5757.598,E2 -5757.598} C_VEL
LIN {X 0,Y 503.025,Z 482.641,A -85,B 0,C 180,E1 -5760,E2 -5760} C_VEL
LIN {X 0,Y 503.023,Z 482.641,A -85,B 0,C 180,E1 -5762.402,E2 -5762.402} C_VEL
LIN {X 0,Y 502.938,Z 482.651,A -85,B 0,C 180,E1 -5765.613,E2 -5765.613} C_VEL
LIN {X 0,Y 502.9,Z 482.656,A -85,B 0,C 180,E1 -5768.033,E2 -5768.033} C_VEL
LIN {X 0,Y 502.876,Z 482.659,A -85,B 0,C 180,E1 -5771.283,E2 -5771.283} C_VEL
LIN {X 0,Y 502.843,Z 482.663,A -85,B 0,C 180,E1 -5774.571,E2 -5774.571} C_VEL
LIN {X 0,Y 502.86,Z 482.663,A -85,B 0,C 180,E1 -5777.907,E2 -5777.907} C_VEL
LIN {X 0,Y 502.826,Z 482.665,A -85,B 0,C 180,E1 -5780.536,E2 -5780.536} C_VEL
LIN {X 0,Y 502.795,Z 482.67,A -85,B 0,C 180,E1 -5783.04,E2 -5783.04} C_VEL
LIN {X 0,Y 502.838,Z 482.663,A -85,B 0,C 180,E1 -5785.676,E2 -5785.676} C_VEL
LIN {X 0,Y 502.84,Z 482.663,A -85,B 0,C 180,E1 -5788.373,E2 -5788.373} C_VEL
LIN {X 0,Y 502.795,Z 482.669,A -85,B 0,C 180,E1 -5791.5,E2 -5791.5} C_VEL
LIN {X 0,Y 502.804,Z 482.668,A -85,B 0,C 180,E1 -5794.445,E2 -5794.445} C_VEL
LIN {X 0,Y 502.779,Z 482.672,A -85,B 0,C 180,E1 -5797.179,E2 -5797.179} C_VEL
LIN {X 0,Y 502.785,Z 482.67,A -85,B 0,C 180,E1 -5800.015,E2 -5800.015} C_VEL
LIN {X 0,Y 502.801,Z 482.667,A -85,B 0,C 180,E1 -5802.2,E2 -5802.2} C_VEL
LIN {X 0,Y 502.798,Z 482.669,A -85,B 0,C 180,E1 -5805.469,E2 -5805.469} C_VEL
LIN {X 0,Y 502.825,Z 482.666,A -85,B 0,C 180,E1 -5809.004,E2 -5809.004} C_VEL
LIN {X 0,Y 502.796,Z 482.67,A -85,B 0,C 180,E1 -5812.047,E2 -5812.047} C_VEL
LIN {X 0,Y 502.809,Z 482.669,A -85,B 0,C 180,E1 -5815.036,E2 -5815.036} C_VEL
LIN {X 0,Y 502.875,Z 482.768,A -85,B 0,C 180,E1 -5816.314,E2 -5816.314} C_VEL
LIN {X 0,Y 503.772,Z 488.193,A -85,B 0,C 180,E1 -5818.32,E2 -5818.32} C_VEL
LIN {X 0,Y 503.721,Z 493.913,A -85,B 0,C 180,E1 -5820.318,E2 -5820.318} C_VEL
LIN {X 0,Y 503.405,Z 502.783,A -85,B 0,C 180,E1 -5823.316,E2 -5823.316} C_VEL
LIN {X 0,Y 503.095,Z 511.27,A -85,B 0,C 180,E1 -5826.102,E2 -5826.102} C_VEL
LIN {X 0,Y 502.86,Z 520.725,A -85,B 0,C 180,E1 -5829.122,E2 -5829.122} C_VEL
LIN {X 0,Y 502.648,Z 530.186,A -85,B 0,C 180,E1 -5832.086,E2 -5832.086} C_VEL
LIN {X 0,Y 502.433,Z 541.062,A -85,B 0,C 180,E1 -5835.417,E2 -5835.417} C_VEL
LIN {X 0,Y 502.335,Z 552.044,A -85,B 0,C 180,E1 -5838.73,E2 -5838.73} C_VEL
LIN {X 0,Y 503.557,Z 563.594,A -85,B 0,C 180,E1 -5839.089,E2 -5839.089} C_VEL
LIN {X 0,Y 503.372,Z 574.022,A -85,B 0,C 180,E1 -5839.543,E2 -5839.543} C_VEL
LIN {X 0,Y 503.215,Z 582.802,A -85,B 0,C 180,E1 -5840.048,E2 -5840.048} C_VEL
LIN {X 0,Y 503.02,Z 591.191,A -85,B 0,C 180,E1 -5840.653,E2 -5840.653} C_VEL
LIN {X 0,Y 502.753,Z 599.129,A -85,B 0,C 180,E1 -5841.358,E2 -5841.358} C_VEL
LIN {X 0,Y 502.575,Z 606.558,A -85,B 0,C 180,E1 -5842.164,E2 -5842.164} C_VEL
LIN {X 0,Y 502.424,Z 613.313,A -85,B 0,C 180,E1 -5843.061,E2 -5843.061} C_VEL
LIN {X 0,Y 502.343,Z 620.037,A -85,B 0,C 180,E1 -5844.179,E2 -5844.179} C_VEL
LIN {X 0,Y 502.154,Z 624.695,A -85,B 0,C 180,E1 -5845.183,E2 -5845.183} C_VEL
LIN {X 0,Y 502.181,Z 627.723,A -85,B 0,C 180,E1 -5845.988,E2 -5845.988} C_VEL
LIN {X 0,Y 502.134,Z 630.065,A -85,B 0,C 180,E1 -5846.791,E2 -5846.791} C_VEL
LIN {X 0,Y 502.122,Z 631.834,A -85,B 0,C 180,E1 -5847.594,E2 -5847.594} C_VEL
LIN {X 0,Y 502.035,Z 633.096,A -85,B 0,C 180,E1 -5848.396,E2 -5848.396} C_VEL
LIN {X 0,Y 501.988,Z 633.878,A -85,B 0,C 180,E1 -5849.198,E2 -5849.198} C_VEL
LIN {X 0,Y 501.977,Z 634.168,A -85,B 0,C 180,E1 -5850,E2 -5850} C_VEL
LIN {X 0,Y 501.988,Z 633.865,A -85,B 0,C 180,E1 -5850.803,E2 -5850.803} C_VEL
LIN {X 0,Y 502.035,Z 633.074,A -85,B 0,C 180,E1 -5851.605,E2 -5851.605} C_VEL
LIN {X 0,Y 502.123,Z 631.796,A -85,B 0,C 180,E1 -5852.407,E2 -5852.407} C_VEL
LIN {X 0,Y 502.173,Z 628.849,A -85,B 0,C 180,E1 -5853.611,E2 -5853.611} C_VEL
LIN {X 0,Y 502.161,Z 626.149,A -85,B 0,C 180,E1 -5854.415,E2 -5854.415} C_VEL
LIN {X 0,Y 502.285,Z 620.889,A -85,B 0,C 180,E1 -5855.621,E2 -5855.621} C_VEL
LIN {X 0,Y 502.412,Z 614.824,A -85,B 0,C 180,E1 -5856.693,E2 -5856.693} C_VEL
LIN {X 0,Y 502.527,Z 608.066,A -85,B 0,C 180,E1 -5857.635,E2 -5857.635} C_VEL
LIN {X 0,Y 502.748,Z 599.906,A -85,B 0,C 180,E1 -5858.542,E2 -5858.542} C_VEL
LIN {X 0,Y 502.973,Z 592.114,A -85,B 0,C 180,E1 -5859.247,E2 -5859.247} C_VEL
LIN {X 0,Y 503.157,Z 583.929,A -85,B 0,C 180,E1 -5859.853,E2 -5859.853} C_VEL
LIN {X 0,Y 503.346,Z 575.457,A -85,B 0,C 180,E1 -5860.357,E2 -5860.357} C_VEL
LIN {X 0,Y 503.549,Z 565.641,A -85,B 0,C 180,E1 -5860.81,E2 -5860.81} C_VEL
LIN {X 0,Y 502.464,Z 554.299,A -85,B 0,C 180,E1 -5861.204,E2 -5861.204} C_VEL
LIN {X 0,Y 502.255,Z 551.947,A -85,B 0,C 180,E1 -5861.272,E2 -5861.272} C_VEL
LIN {X 0,Y 502.37,Z 541.419,A -85,B 0,C 180,E1 -5864.585,E2 -5864.585} C_VEL
LIN {X 0,Y 502.481,Z 532.241,A -85,B 0,C 180,E1 -5867.501,E2 -5867.501} C_VEL
LIN {X 0,Y 502.643,Z 524.435,A -85,B 0,C 180,E1 -5870.033,E2 -5870.033} C_VEL
LIN {X 0,Y 502.874,Z 514.169,A -85,B 0,C 180,E1 -5873.473,E2 -5873.473} C_VEL
LIN {X 0,Y 503.055,Z 506.672,A -85,B 0,C 180,E1 -5876.109,E2 -5876.109} C_VEL
LIN {X 0,Y 503.352,Z 499.444,A -85,B 0,C 180,E1 -5878.797,E2 -5878.797} C_VEL
LIN {X 0,Y 503.827,Z 491.529,A -85,B 0,C 180,E1 -5882.011,E2 -5882.011} C_VEL
LIN {X 0,Y 503.824,Z 488.929,A -85,B 0,C 180,E1 -5883.18,E2 -5883.18} C_VEL
LIN {X 0,Y 503.002,Z 483.659,A -85,B 0,C 180,E1 -5885.933,E2 -5885.933} C_VEL
LIN {X 0,Y 502.807,Z 482.669,A -85,B 0,C 180,E1 -5886.57,E2 -5886.57} C_VEL
LIN {X 0,Y 502.791,Z 482.671,A -85,B 0,C 180,E1 -5889.755,E2 -5889.755} C_VEL
LIN {X 0,Y 502.805,Z 482.668,A -85,B 0,C 180,E1 -5892.199,E2 -5892.199} C_VEL
LIN {X 0,Y 502.803,Z 482.667,A -85,B 0,C 180,E1 -5895.468,E2 -5895.468} C_VEL
LIN {X 0,Y 502.833,Z 482.665,A -85,B 0,C 180,E1 -5897.865,E2 -5897.865} C_VEL
LIN {X 0,Y 502.804,Z 482.669,A -85,B 0,C 180,E1 -5901.024,E2 -5901.024} C_VEL
LIN {X 0,Y 502.777,Z 482.672,A -85,B 0,C 180,E1 -5904.169,E2 -5904.169} C_VEL
LIN {X 0,Y 502.77,Z 482.673,A -85,B 0,C 180,E1 -5907.005,E2 -5907.005} C_VEL
LIN {X 0,Y 502.729,Z 482.793,A -85,B 0,C 180,E1 -5907.912,E2 -5907.912} C_VEL
LIN {X 0,Y 502.622,Z 485.818,A -85,B 0,C 180,E1 -5910.699,E2 -5910.699} C_VEL
LIN {X 0,Y 502.521,Z 489.058,A -85,B 0,C 180,E1 -5913.518,E2 -5913.518} C_VEL
LIN {X 0,Y 502.409,Z 492.091,A -85,B 0,C 180,E1 -5916.067,E2 -5916.067} C_VEL
LIN {X 0,Y 502.355,Z 495.269,A -85,B 0,C 180,E1 -5918.67,E2 -5918.67} C_VEL
LIN {X 0,Y 502.256,Z 498.487,A -85,B 0,C 180,E1 -5921.226,E2 -5921.226} C_VEL
LIN {X 0,Y 502.237,Z 501.719,A -85,B 0,C 180,E1 -5923.748,E2 -5923.748} C_VEL
LIN {X 0,Y 502.167,Z 504.973,A -85,B 0,C 180,E1 -5926.236,E2 -5926.236} C_VEL
LIN {X 0,Y 502.176,Z 508.449,A -85,B 0,C 180,E1 -5928.854,E2 -5928.854} C_VEL
LIN {X 0,Y 503.601,Z 518.605,A -85,B 0,C 180,E1 -5929.242,E2 -5929.242} C_VEL
LIN {X 0,Y 503.497,Z 527.404,A -85,B 0,C 180,E1 -5929.647,E2 -5929.647} C_VEL
LIN {X 0,Y 503.284,Z 535.956,A -85,B 0,C 180,E1 -5930.15,E2 -5930.15} C_VEL
LIN {X 0,Y 503.101,Z 544.161,A -85,B 0,C 180,E1 -5930.756,E2 -5930.756} C_VEL
LIN {X 0,Y 502.904,Z 551.947,A -85,B 0,C 180,E1 -5931.461,E2 -5931.461} C_VEL
LIN {X 0,Y 502.689,Z 558.382,A -85,B 0,C 180,E1 -5932.166,E2 -5932.166} C_VEL
LIN {X 0,Y 502.553,Z 564.535,A -85,B 0,C 180,E1 -5932.976,E2 -5932.976} C_VEL
LIN {X 0,Y 502.463,Z 570.747,A -85,B 0,C 180,E1 -5933.978,E2 -5933.978} C_VEL
LIN {X 0,Y 502.203,Z 576.56,A -85,B 0,C 180,E1 -5935.183,E2 -5935.183} C_VEL
LIN {X 0,Y 502.256,Z 579.556,A -85,B 0,C 180,E1 -5935.988,E2 -5935.988} C_VEL
LIN {X 0,Y 502.149,Z 581.889,A -85,B 0,C 180,E1 -5936.791,E2 -5936.791} C_VEL
LIN {X 0,Y 502.124,Z 583.67,A -85,B 0,C 180,E1 -5937.594,E2 -5937.594} C_VEL
LIN {X 0,Y 502.037,Z 584.957,A -85,B 0,C 180,E1 -5938.396,E2 -5938.396} C_VEL
LIN {X 0,Y 501.989,Z 585.766,A -85,B 0,C 180,E1 -5939.198,E2 -5939.198} C_VEL
LIN {X 0,Y 501.978,Z 586.065,A -85,B 0,C 180,E1 -5940,E2 -5940} C_VEL
LIN {X 0,Y 501.99,Z 585.785,A -85,B 0,C 180,E1 -5940.802,E2 -5940.802} C_VEL
LIN {X 0,Y 502.036,Z 585.037,A -85,B 0,C 180,E1 -5941.604,E2 -5941.604} C_VEL
LIN {X 0,Y 502.122,Z 583.806,A -85,B 0,C 180,E1 -5942.407,E2 -5942.407} C_VEL
LIN {X 0,Y 502.172,Z 580.938,A -85,B 0,C 180,E1 -5943.611,E2 -5943.611} C_VEL
LIN {X 0,Y 502.245,Z 578.317,A -85,B 0,C 180,E1 -5944.414,E2 -5944.414} C_VEL
LIN {X 0,Y 502.336,Z 573.176,A -85,B 0,C 180,E1 -5945.62,E2 -5945.62} C_VEL
LIN {X 0,Y 502.524,Z 568.262,A -85,B 0,C 180,E1 -5946.519,E2 -5946.519} C_VEL
LIN {X 0,Y 502.621,Z 560.671,A -85,B 0,C 180,E1 -5947.634,E2 -5947.634} C_VEL
LIN {X 0,Y 502.87,Z 552.68,A -85,B 0,C 180,E1 -5948.54,E2 -5948.54} C_VEL
LIN {X 0,Y 503.104,Z 545.061,A -85,B 0,C 180,E1 -5949.244,E2 -5949.244} C_VEL
LIN {X 0,Y 503.289,Z 537.074,A -85,B 0,C 180,E1 -5949.85,E2 -5949.85} C_VEL
LIN {X 0,Y 503.485,Z 528.822,A -85,B 0,C 180,E1 -5950.353,E2 -5950.353} C_VEL
LIN {X 0,Y 503.59,Z 520.464,A -85,B 0,C 180,E1 -5950.758,E2 -5950.758} C_VEL
LIN {X 0,Y 503.1,Z 513.93,A -85,B 0,C 180,E1 -5951.023,E2 -5951.023} C_VEL
LIN {X 0,Y 502.199,Z 507.729,A -85,B 0,C 180,E1 -5951.248,E2 -5951.248} C_VEL
LIN {X 0,Y 502.172,Z 502.781,A -85,B 0,C 180,E1 -5954.591,E2 -5954.591} C_VEL
LIN {X 0,Y 502.233,Z 497.851,A -85,B 0,C 180,E1 -5957.93,E2 -5957.93} C_VEL
LIN {X 0,Y 502.265,Z 494.203,A -85,B 0,C 180,E1 -5960.476,E2 -5960.476} C_VEL
LIN {X 0,Y 502.263,Z 490.478,A -85,B 0,C 180,E1 -5963.066,E2 -5963.066} C_VEL
LIN {X 0,Y 502.346,Z 486.768,A -85,B 0,C 180,E1 -5965.703,E2 -5965.703} C_VEL
LIN {X 0,Y 502.501,Z 484.707,A -85,B 0,C 180,E1 -5967.261,E2 -5967.261} C_VEL
LIN {X 0,Y 502.477,Z 489.602,A -85,B 0,C 180,E1 -5969.31,E2 -5969.31} C_VEL
LIN {X 0,Y 502.512,Z 496.292,A -85,B 0,C 180,E1 -5972.104,E2 -5972.104} C_VEL
LIN {X 0,Y 502.463,Z 501.658,A -85,B 0,C 180,E1 -5974.387,E2 -5974.387} C_VEL
LIN {X 0,Y 502.364,Z 508.96,A -85,B 0,C 180,E1 -5977.519,E2 -5977.519} C_VEL
LIN {X 0,Y 502.289,Z 514.81,A -85,B 0,C 180,E1 -5980.063,E2 -5980.063} C_VEL
LIN {X 0,Y 502.236,Z 522.268,A -85,B 0,C 180,E1 -5983.309,E2 -5983.309} C_VEL
LIN {X 0,Y 502.224,Z 525.819,A -85,B 0,C 180,E1 -5984.814,E2 -5984.814} C_VEL
LIN {X 0,Y 503.56,Z 535.315,A -85,B 0,C 180,E1 -5985.127,E2 -5985.127} C_VEL
LIN {X 0,Y 503.53,Z 545.516,A -85,B 0,C 180,E1 -5985.559,E2 -5985.559} C_VEL
LIN {X 0,Y 503.269,Z 556.331,A -85,B 0,C 180,E1 -5986.194,E2 -5986.194} C_VEL
LIN {X 0,Y 503.014,Z 564.317,A -85,B 0,C 180,E1 -5986.794,E2 -5986.794} C_VEL
LIN {X 0,Y 502.817,Z 571.537,A -85,B 0,C 180,E1 -5987.457,E2 -5987.457} C_VEL
LIN {X 0,Y 502.652,Z 578.33,A -85,B 0,C 180,E1 -5988.21,E2 -5988.21} C_VEL
LIN {X 0,Y 501.841,Z 582.352,A -85,B 0,C 180,E1 -5988.708,E2 -5988.708} C_VEL
LIN {X 0,Y 498.816,Z 588.235,A -85,B 0,C 180,E1 -5989.557,E2 -5989.557} C_VEL
LIN {X 0,Y 495.848,Z 593.369,A -85,B 0,C 180,E1 -5990.473,E2 -5990.473} C_VEL
LIN {X 0,Y 495.121,Z 596.065,A -85,B 0,C 180,E1 -5991.068,E2 -5991.068} C_VEL
LIN {X 0,Y 495.044,Z 600.542,A -85,B 0,C 180,E1 -5992.377,E2 -5992.377} C_VEL
LIN {X 0,Y 494.946,Z 603.014,A -85,B 0,C 180,E1 -5993.388,E2 -5993.388} C_VEL
LIN {X 0,Y 494.929,Z 604.654,A -85,B 0,C 180,E1 -5994.394,E2 -5994.394} C_VEL
LIN {X 0,Y 494.912,Z 605.539,A -85,B 0,C 180,E1 -5995.45,E2 -5995.45} C_VEL
LIN {X 0,Y 494.88,Z 605.429,A -85,B 0,C 180,E1 -5996.917,E2 -5996.917} C_VEL
LIN {X 0,Y 494.965,Z 603.538,A -85,B 0,C 180,E1 -5998.423,E2 -5998.423} C_VEL
LIN {X 0,Y 495.038,Z 600.663,A -85,B 0,C 180,E1 -5999.662,E2 -5999.662} C_VEL
LIN {X 0,Y 495.098,Z 597.334,A -85,B 0,C 180,E1 -6000.677,E2 -6000.677} C_VEL
LIN {X 0,Y 495.19,Z 592.253,A -85,B 0,C 180,E1 -6001.857,E2 -6001.857} C_VEL
LIN {X 0,Y 495.413,Z 585.669,A -85,B 0,C 180,E1 -6003.002,E2 -6003.002} C_VEL
LIN {X 0,Y 495.545,Z 579.077,A -85,B 0,C 180,E1 -6003.918,E2 -6003.918} C_VEL
LIN {X 0,Y 495.792,Z 572.012,A -85,B 0,C 180,E1 -6004.72,E2 -6004.72} C_VEL
LIN {X 0,Y 496.08,Z 563.074,A -85,B 0,C 180,E1 -6005.545,E2 -6005.545} C_VEL
LIN {X 0,Y 496.345,Z 552.202,A -85,B 0,C 180,E1 -6006.31,E2 -6006.31} C_VEL
LIN {X 0,Y 496.558,Z 543.505,A -85,B 0,C 180,E1 -6006.778,E2 -6006.778} C_VEL
LIN {X 0,Y 496.524,Z 536.159,A -85,B 0,C 180,E1 -6007.093,E2 -6007.093} C_VEL
LIN {X 0,Y 495.076,Z 526.011,A -85,B 0,C 180,E1 -6007.462,E2 -6007.462} C_VEL
LIN {X 0,Y 495.13,Z 520.448,A -85,B 0,C 180,E1 -6010.082,E2 -6010.082} C_VEL
LIN {X 0,Y 495.182,Z 514.953,A -85,B 0,C 180,E1 -6012.659,E2 -6012.659} C_VEL
LIN {X 0,Y 495.252,Z 509.534,A -85,B 0,C 180,E1 -6015.2,E2 -6015.2} C_VEL
LIN {X 0,Y 495.387,Z 502.384,A -85,B 0,C 180,E1 -6018.544,E2 -6018.544} C_VEL
LIN {X 0,Y 495.409,Z 495.294,A -85,B 0,C 180,E1 -6021.844,E2 -6021.844} C_VEL
LIN {X 0,Y 495.435,Z 489.941,A -85,B 0,C 180,E1 -6024.301,E2 -6024.301} C_VEL
LIN {X 0,Y 495.506,Z 486.384,A -85,B 0,C 180,E1 -6025.933,E2 -6025.933} C_VEL
LIN {X 0,Y 495.456,Z 483.584,A -85,B 0,C 180,E1 -6027.256,E2 -6027.256} C_VEL
LIN {X 0,Y 495.939,Z 483.523,A -85,B 0,C 180,E1 -6029.188,E2 -6029.188} C_VEL
LIN {X 0,Y 496.007,Z 483.514,A -85,B 0,C 180,E1 -6030.811,E2 -6030.811} C_VEL
LIN {X 0,Y 495.843,Z 483.534,A -85,B 0,C 180,E1 -6033.25,E2 -6033.25} C_VEL
LIN {X 0,Y 495.883,Z 483.531,A -85,B 0,C 180,E1 -6036.51,E2 -6036.51} C_VEL
LIN {X 0,Y 495.841,Z 483.534,A -85,B 0,C 180,E1 -6038.969,E2 -6038.969} C_VEL
LIN {X 0,Y 495.83,Z 483.536,A -85,B 0,C 180,E1 -6042.034,E2 -6042.034} C_VEL
LIN {X 0,Y 495.825,Z 483.535,A -85,B 0,C 180,E1 -6045.451,E2 -6045.451} C_VEL
LIN {X 0,Y 495.807,Z 483.542,A -85,B 0,C 180,E1 -6048.247,E2 -6048.247} C_VEL
LIN {X 0,Y 495.775,Z 483.543,A -85,B 0,C 180,E1 -6050.756,E2 -6050.756} C_VEL
LIN {X 0,Y 495.753,Z 483.545,A -85,B 0,C 180,E1 -6053.386,E2 -6053.386} C_VEL
LIN {X 0,Y 495.8,Z 483.54,A -85,B 0,C 180,E1 -6056.067,E2 -6056.067} C_VEL
LIN {X 0,Y 495.779,Z 483.543,A -85,B 0,C 180,E1 -6058.814,E2 -6058.814} C_VEL
LIN {X 0,Y 495.759,Z 483.545,A -85,B 0,C 180,E1 -6061.726,E2 -6061.726} C_VEL
LIN {X 0,Y 495.776,Z 483.544,A -85,B 0,C 180,E1 -6064.695,E2 -6064.695} C_VEL
LIN {X 0,Y 495.731,Z 483.549,A -85,B 0,C 180,E1 -6067.561,E2 -6067.561} C_VEL
LIN {X 0,Y 495.765,Z 483.545,A -85,B 0,C 180,E1 -6070.699,E2 -6070.699} C_VEL
LIN {X 0,Y 495.733,Z 483.548,A -85,B 0,C 180,E1 -6073.695,E2 -6073.695} C_VEL
LIN {X 0,Y 495.733,Z 483.549,A -85,B 0,C 180,E1 -6076.304,E2 -6076.304} C_VEL
LIN {X 0,Y 495.779,Z 483.543,A -85,B 0,C 180,E1 -6079.301,E2 -6079.301} C_VEL
LIN {X 0,Y 495.729,Z 483.55,A -85,B 0,C 180,E1 -6082.438,E2 -6082.438} C_VEL
LIN {X 0,Y 495.776,Z 483.543,A -85,B 0,C 180,E1 -6085.457,E2 -6085.457} C_VEL
LIN {X 0,Y 495.757,Z 483.547,A -85,B 0,C 180,E1 -6088.364,E2 -6088.364} C_VEL
LIN {X 0,Y 495.786,Z 483.541,A -85,B 0,C 180,E1 -6091.506,E2 -6091.506} C_VEL
LIN {X 0,Y 495.798,Z 483.541,A -85,B 0,C 180,E1 -6093.932,E2 -6093.932} C_VEL
LIN {X 0,Y 495.763,Z 483.544,A -85,B 0,C 180,E1 -6097.137,E2 -6097.137} C_VEL
LIN {X 0,Y 495.776,Z 483.545,A -85,B 0,C 180,E1 -6100.11,E2 -6100.11} C_VEL
LIN {X 0,Y 495.785,Z 483.542,A -85,B 0,C 180,E1 -6102.681,E2 -6102.681} C_VEL
LIN {X 0,Y 495.788,Z 483.542,A -85,B 0,C 180,E1 -6105.217,E2 -6105.217} C_VEL
LIN {X 0,Y 495.866,Z 483.532,A -85,B 0,C 180,E1 -6108.555,E2 -6108.555} C_VEL
LIN {X 0,Y 495.871,Z 483.532,A -85,B 0,C 180,E1 -6111.852,E2 -6111.852} C_VEL
LIN {X 0,Y 495.894,Z 483.53,A -85,B 0,C 180,E1 -6114.306,E2 -6114.306} C_VEL
LIN {X 0,Y 495.993,Z 483.516,A -85,B 0,C 180,E1 -6117.564,E2 -6117.564} C_VEL
LIN {X 0,Y 495.996,Z 483.516,A -85,B 0,C 180,E1 -6120,E2 -6120} C_VEL
LIN {X 0,Y 495.991,Z 483.517,A -85,B 0,C 180,E1 -6122.436,E2 -6122.436} C_VEL
LIN {X 0,Y 495.896,Z 483.528,A -85,B 0,C 180,E1 -6125.693,E2 -6125.693} C_VEL
LIN {X 0,Y 495.871,Z 483.531,A -85,B 0,C 180,E1 -6128.148,E2 -6128.148} C_VEL
LIN {X 0,Y 495.85,Z 483.534,A -85,B 0,C 180,E1 -6131.445,E2 -6131.445} C_VEL
LIN {X 0,Y 495.788,Z 483.542,A -85,B 0,C 180,E1 -6134.783,E2 -6134.783} C_VEL
LIN {X 0,Y 495.786,Z 483.542,A -85,B 0,C 180,E1 -6137.319,E2 -6137.319} C_VEL
LIN {X 0,Y 495.776,Z 483.543,A -85,B 0,C 180,E1 -6139.89,E2 -6139.89} C_VEL
LIN {X 0,Y 495.756,Z 483.546,A -85,B 0,C 180,E1 -6142.861,E2 -6142.861} C_VEL
LIN {X 0,Y 495.788,Z 483.543,A -85,B 0,C 180,E1 -6146.068,E2 -6146.068} C_VEL
LIN {X 0,Y 495.778,Z 483.543,A -85,B 0,C 180,E1 -6148.814,E2 -6148.814} C_VEL
LIN {X 0,Y 495.757,Z 483.546,A -85,B 0,C 180,E1 -6151.726,E2 -6151.726} C_VEL
LIN {X 0,Y 495.774,Z 483.544,A -85,B 0,C 180,E1 -6154.696,E2 -6154.696} C_VEL
LIN {X 0,Y 495.729,Z 483.549,A -85,B 0,C 180,E1 -6157.562,E2 -6157.562} C_VEL
LIN {X 0,Y 495.764,Z 483.545,A -85,B 0,C 180,E1 -6160.7,E2 -6160.7} C_VEL
LIN {X 0,Y 495.733,Z 483.549,A -85,B 0,C 180,E1 -6163.696,E2 -6163.696} C_VEL
LIN {X 0,Y 495.726,Z 483.55,A -85,B 0,C 180,E1 -6166.306,E2 -6166.306} C_VEL
LIN {X 0,Y 495.779,Z 483.543,A -85,B 0,C 180,E1 -6169.302,E2 -6169.302} C_VEL
LIN {X 0,Y 495.762,Z 483.546,A -85,B 0,C 180,E1 -6171.41,E2 -6171.41} C_VEL
LIN {X 0,Y 495.757,Z 483.547,A -85,B 0,C 180,E1 -6174.464,E2 -6174.464} C_VEL
LIN {X 0,Y 495.811,Z 483.681,A -85,B 0,C 180,E1 -6176.135,E2 -6176.135} C_VEL
LIN {X 0,Y 496.829,Z 489.82,A -85,B 0,C 180,E1 -6178.441,E2 -6178.441} C_VEL
LIN {X 0,Y 496.653,Z 496.468,A -85,B 0,C 180,E1 -6180.778,E2 -6180.778} C_VEL
LIN {X 0,Y 496.343,Z 504.549,A -85,B 0,C 180,E1 -6183.54,E2 -6183.54} C_VEL
LIN {X 0,Y 496.028,Z 513.834,A -85,B 0,C 180,E1 -6186.627,E2 -6186.627} C_VEL
LIN {X 0,Y 495.76,Z 523.366,A -85,B 0,C 180,E1 -6189.716,E2 -6189.716} C_VEL
LIN {X 0,Y 495.482,Z 534.049,A -85,B 0,C 180,E1 -6193.096,E2 -6193.096} C_VEL
LIN {X 0,Y 495.312,Z 543.56,A -85,B 0,C 180,E1 -6196.042,E2 -6196.042} C_VEL
LIN {X 0,Y 495.269,Z 551.744,A -85,B 0,C 180,E1 -6198.568,E2 -6198.568} C_VEL
LIN {X 0,Y 496.566,Z 564.473,A -85,B 0,C 180,E1 -6198.985,E2 -6198.985} C_VEL
LIN {X 0,Y 496.347,Z 575.47,A -85,B 0,C 180,E1 -6199.497,E2 -6199.497} C_VEL
LIN {X 0,Y 496.143,Z 583.886,A -85,B 0,C 180,E1 -6200.008,E2 -6200.008} C_VEL
LIN {X 0,Y 495.959,Z 592.011,A -85,B 0,C 180,E1 -6200.622,E2 -6200.622} C_VEL
LIN {X 0,Y 495.701,Z 599.751,A -85,B 0,C 180,E1 -6201.336,E2 -6201.336} C_VEL
LIN {X 0,Y 495.458,Z 607.877,A -85,B 0,C 180,E1 -6202.256,E2 -6202.256} C_VEL
LIN {X 0,Y 495.279,Z 615.504,A -85,B 0,C 180,E1 -6203.362,E2 -6203.362} C_VEL
LIN {X 0,Y 495.218,Z 620.647,A -85,B 0,C 180,E1 -6204.299,E2 -6204.299} C_VEL
LIN {X 0,Y 495.062,Z 625.876,A -85,B 0,C 180,E1 -6205.522,E2 -6205.522} C_VEL
LIN {X 0,Y 495.092,Z 628.562,A -85,B 0,C 180,E1 -6206.338,E2 -6206.338} C_VEL
LIN {X 0,Y 495.026,Z 631.495,A -85,B 0,C 180,E1 -6207.559,E2 -6207.559} C_VEL
LIN {X 0,Y 494.962,Z 632.761,A -85,B 0,C 180,E1 -6208.373,E2 -6208.373} C_VEL
LIN {X 0,Y 494.908,Z 633.543,A -85,B 0,C 180,E1 -6209.187,E2 -6209.187} C_VEL
LIN {X 0,Y 494.895,Z 633.83,A -85,B 0,C 180,E1 -6210,E2 -6210} C_VEL
LIN {X 0,Y 494.908,Z 633.523,A -85,B 0,C 180,E1 -6210.814,E2 -6210.814} C_VEL
LIN {X 0,Y 494.962,Z 632.728,A -85,B 0,C 180,E1 -6211.628,E2 -6211.628} C_VEL
LIN {X 0,Y 495.027,Z 631.443,A -85,B 0,C 180,E1 -6212.441,E2 -6212.441} C_VEL
LIN {X 0,Y 495.096,Z 628.479,A -85,B 0,C 180,E1 -6213.663,E2 -6213.663} C_VEL
LIN {X 0,Y 495.078,Z 624.211,A -85,B 0,C 180,E1 -6214.886,E2 -6214.886} C_VEL
LIN {X 0,Y 495.263,Z 618.379,A -85,B 0,C 180,E1 -6216.11,E2 -6216.11} C_VEL
LIN {X 0,Y 495.377,Z 612.068,A -85,B 0,C 180,E1 -6217.131,E2 -6217.131} C_VEL
LIN {X 0,Y 495.516,Z 605.895,A -85,B 0,C 180,E1 -6217.949,E2 -6217.949} C_VEL
LIN {X 0,Y 495.715,Z 598.391,A -85,B 0,C 180,E1 -6218.767,E2 -6218.767} C_VEL
LIN {X 0,Y 495.977,Z 590.369,A -85,B 0,C 180,E1 -6219.482,E2 -6219.482} C_VEL
LIN {X 0,Y 496.206,Z 580.385,A -85,B 0,C 180,E1 -6220.198,E2 -6220.198} C_VEL
LIN {X 0,Y 496.452,Z 569.824,A -85,B 0,C 180,E1 -6220.76,E2 -6220.76} C_VEL
LIN {X 0,Y 496.314,Z 562.46,A -85,B 0,C 180,E1 -6221.073,E2 -6221.073} C_VEL
LIN {X 0,Y 495.168,Z 551.543,A -85,B 0,C 180,E1 -6221.436,E2 -6221.436} C_VEL
LIN {X 0,Y 495.306,Z 541.021,A -85,B 0,C 180,E1 -6224.798,E2 -6224.798} C_VEL
LIN {X 0,Y 495.464,Z 530.781,A -85,B 0,C 180,E1 -6228.126,E2 -6228.126} C_VEL
LIN {X 0,Y 495.615,Z 521.579,A -85,B 0,C 180,E1 -6231.199,E2 -6231.199} C_VEL
LIN {X 0,Y 495.826,Z 513.965,A -85,B 0,C 180,E1 -6233.827,E2 -6233.827} C_VEL
LIN {X 0,Y 496.118,Z 505.37,A -85,B 0,C 180,E1 -6236.957,E2 -6236.957} C_VEL
LIN {X 0,Y 496.463,Z 498.32,A -85,B 0,C 180,E1 -6239.701,E2 -6239.701} C_VEL
LIN {X 0,Y 496.881,Z 491.738,A -85,B 0,C 180,E1 -6242.513,E2 -6242.513} C_VEL
LIN {X 0,Y 496.494,Z 487.748,A -85,B 0,C 180,E1 -6244.487,E2 -6244.487} C_VEL
LIN {X 0,Y 495.758,Z 483.548,A -85,B 0,C 180,E1 -6246.985,E2 -6246.985} C_VEL
LIN {X 0,Y 495.761,Z 483.547,A -85,B 0,C 180,E1 -6250.047,E2 -6250.047} C_VEL
LIN {X 0,Y 495.729,Z 483.549,A -85,B 0,C 180,E1 -6252.883,E2 -6252.883} C_VEL
LIN {X 0,Y 495.74,Z 483.547,A -85,B 0,C 180,E1 -6256,E2 -6256} C_VEL
LIN {X 0,Y 495.766,Z 483.545,A -85,B 0,C 180,E1 -6258.706,E2 -6258.706} C_VEL
LIN {X 0,Y 495.753,Z 483.548,A -85,B 0,C 180,E1 -6261.409,E2 -6261.409} C_VEL
LIN {X 0,Y 495.75,Z 483.548,A -85,B 0,C 180,E1 -6264.463,E2 -6264.463} C_VEL
LIN {X 0,Y 495.691,Z 483.556,A -85,B 0,C 180,E1 -6267.4,E2 -6267.4} C_VEL
LIN {X 0,Y 495.665,Z 485.3,A -85,B 0,C 180,E1 -6269.307,E2 -6269.307} C_VEL
LIN {X 0,Y 495.528,Z 488.34,A -85,B 0,C 180,E1 -6272.093,E2 -6272.093} C_VEL
LIN {X 0,Y 495.43,Z 491.912,A -85,B 0,C 180,E1 -6275.215,E2 -6275.215} C_VEL
LIN {X 0,Y 495.305,Z 495.668,A -85,B 0,C 180,E1 -6278.351,E2 -6278.351} C_VEL
LIN {X 0,Y 495.215,Z 498.868,A -85,B 0,C 180,E1 -6280.949,E2 -6280.949} C_VEL
LIN {X 0,Y 495.18,Z 503.185,A -85,B 0,C 180,E1 -6284.356,E2 -6284.356} C_VEL
LIN {X 0,Y 495.087,Z 507.551,A -85,B 0,C 180,E1 -6287.706,E2 -6287.706} C_VEL
LIN {X 0,Y 495.136,Z 508.851,A -85,B 0,C 180,E1 -6288.694,E2 -6288.694} C_VEL
LIN {X 0,Y 496.602,Z 518.814,A -85,B 0,C 180,E1 -6289.089,E2 -6289.089} C_VEL
LIN {X 0,Y 496.522,Z 527.625,A -85,B 0,C 180,E1 -6289.5,E2 -6289.5} C_VEL
LIN {X 0,Y 496.296,Z 536.187,A -85,B 0,C 180,E1 -6290.01,E2 -6290.01} C_VEL
LIN {X 0,Y 496.116,Z 544.409,A -85,B 0,C 180,E1 -6290.624,E2 -6290.624} C_VEL
LIN {X 0,Y 495.903,Z 552.213,A -85,B 0,C 180,E1 -6291.34,E2 -6291.34} C_VEL
LIN {X 0,Y 495.676,Z 558.665,A -85,B 0,C 180,E1 -6292.054,E2 -6292.054} C_VEL
LIN {X 0,Y 495.509,Z 565.062,A -85,B 0,C 180,E1 -6292.909,E2 -6292.909} C_VEL
LIN {X 0,Y 495.365,Z 572.198,A -85,B 0,C 180,E1 -6294.096,E2 -6294.096} C_VEL
LIN {X 0,Y 495.127,Z 576.89,A -85,B 0,C 180,E1 -6295.114,E2 -6295.114} C_VEL
LIN {X 0,Y 495.193,Z 579.89,A -85,B 0,C 180,E1 -6295.931,E2 -6295.931} C_VEL
LIN {X 0,Y 495.072,Z 582.227,A -85,B 0,C 180,E1 -6296.745,E2 -6296.745} C_VEL
LIN {X 0,Y 495.058,Z 584.011,A -85,B 0,C 180,E1 -6297.559,E2 -6297.559} C_VEL
LIN {X 0,Y 494.964,Z 585.3,A -85,B 0,C 180,E1 -6298.373,E2 -6298.373} C_VEL
LIN {X 0,Y 494.909,Z 586.11,A -85,B 0,C 180,E1 -6299.186,E2 -6299.186} C_VEL
LIN {X 0,Y 494.896,Z 586.405,A -85,B 0,C 180,E1 -6300,E2 -6300} C_VEL
LIN {X 0,Y 494.91,Z 586.121,A -85,B 0,C 180,E1 -6300.814,E2 -6300.814} C_VEL
LIN {X 0,Y 494.963,Z 585.366,A -85,B 0,C 180,E1 -6301.627,E2 -6301.627} C_VEL
LIN {X 0,Y 495.056,Z 584.13,A -85,B 0,C 180,E1 -6302.441,E2 -6302.441} C_VEL
LIN {X 0,Y 495.102,Z 581.246,A -85,B 0,C 180,E1 -6303.662,E2 -6303.662} C_VEL
LIN {X 0,Y 495.174,Z 578.618,A -85,B 0,C 180,E1 -6304.477,E2 -6304.477} C_VEL
LIN {X 0,Y 495.293,Z 573.454,A -85,B 0,C 180,E1 -6305.7,E2 -6305.7} C_VEL
LIN {X 0,Y 495.451,Z 567.422,A -85,B 0,C 180,E1 -6306.803,E2 -6306.803} C_VEL
LIN {X 0,Y 495.629,Z 559.216,A -85,B 0,C 180,E1 -6307.947,E2 -6307.947} C_VEL
LIN {X 0,Y 495.874,Z 551.874,A -85,B 0,C 180,E1 -6308.764,E2 -6308.764} C_VEL
LIN {X 0,Y 496.138,Z 544.029,A -85,B 0,C 180,E1 -6309.478,E2 -6309.478} C_VEL
LIN {X 0,Y 496.339,Z 535.762,A -85,B 0,C 180,E1 -6310.092,E2 -6310.092} C_VEL
LIN {X 0,Y 496.584,Z 525.267,A -85,B 0,C 180,E1 -6310.705,E2 -6310.705} C_VEL
LIN {X 0,Y 496.426,Z 517.068,A -85,B 0,C 180,E1 -6311.07,E2 -6311.07} C_VEL
LIN {X 0,Y 495.131,Z 507.999,A -85,B 0,C 180,E1 -6311.41,E2 -6311.41} C_VEL
LIN {X 0,Y 495.135,Z 502.484,A -85,B 0,C 180,E1 -6315.159,E2 -6315.159} C_VEL
LIN {X 0,Y 495.163,Z 498.061,A -85,B 0,C 180,E1 -6318.195,E2 -6318.195} C_VEL
LIN {X 0,Y 495.186,Z 494.372,A -85,B 0,C 180,E1 -6320.782,E2 -6320.782} C_VEL
LIN {X 0,Y 495.205,Z 490.649,A -85,B 0,C 180,E1 -6323.414,E2 -6323.414} C_VEL
LIN {X 0,Y 495.309,Z 486.892,A -85,B 0,C 180,E1 -6326.095,E2 -6326.095} C_VEL
LIN {X 0,Y 495.414,Z 485.355,A -85,B 0,C 180,E1 -6327.226,E2 -6327.226} C_VEL
LIN {X 0,Y 495.419,Z 490.363,A -85,B 0,C 180,E1 -6329.302,E2 -6329.302} C_VEL
LIN {X 0,Y 495.442,Z 497.056,A -85,B 0,C 180,E1 -6332.137,E2 -6332.137} C_VEL
LIN {X 0,Y 495.361,Z 502.859,A -85,B 0,C 180,E1 -6334.625,E2 -6334.625} C_VEL
LIN {X 0,Y 495.287,Z 509.757,A -85,B 0,C 180,E1 -6337.601,E2 -6337.601} C_VEL
LIN {X 0,Y 495.231,Z 515.203,A -85,B 0,C 180,E1 -6339.974,E2 -6339.974} C_VEL
LIN {X 0,Y 495.181,Z 521.97,A -85,B 0,C 180,E1 -6342.942,E2 -6342.942} C_VEL
LIN {X 0,Y 495.135,Z 525.854,A -85,B 0,C 180,E1 -6344.646,E2 -6344.646} C_VEL
LIN {X 0,Y 496.636,Z 536.356,A -85,B 0,C 180,E1 -6345.005,E2 -6345.005} C_VEL
LIN {X 0,Y 496.518,Z 547.766,A -85,B 0,C 180,E1 -6345.52,E2 -6345.52} C_VEL
LIN {X 0,Y 496.266,Z 556.555,A -85,B 0,C 180,E1 -6346.058,E2 -6346.058} C_VEL
LIN {X 0,Y 495.983,Z 565.231,A -85,B 0,C 180,E1 -6346.727,E2 -6346.727} C_VEL
LIN {X 0,Y 495.738,Z 573.238,A -85,B 0,C 180,E1 -6347.493,E2 -6347.493} C_VEL
LIN {X 0,Y 495.552,Z 580.565,A -85,B 0,C 180,E1 -6348.353,E2 -6348.353} C_VEL
LIN {X 0,Y 495.305,Z 588.058,A -85,B 0,C 180,E1 -6349.462,E2 -6349.462} C_VEL
LIN {X 0,Y 495.182,Z 593.827,A -85,B 0,C 180,E1 -6350.57,E2 -6350.57} C_VEL
LIN {X 0,Y 495.121,Z 596.065,A -85,B 0,C 180,E1 -6351.068,E2 -6351.068} C_VEL
LIN {X 0,Y 494.388,Z 598.544,A -85,B 0,C 180,E1 -6351.683,E2 -6351.683} C_VEL
LIN {X 0,Y 492.743,Z 600.582,A -85,B 0,C 180,E1 -6352.302,E2 -6352.302} C_VEL
LIN {X 0,Y 488.953,Z 603.605,A -85,B 0,C 180,E1 -6353.581,E2 -6353.581} C_VEL
LIN {X 0,Y 487.901,Z 604.715,A -85,B 0,C 180,E1 -6354.257,E2 -6354.257} C_VEL
LIN {X 0,Y 487.819,Z 604.933,A -85,B 0,C 180,E1 -6354.487,E2 -6354.487} C_VEL
LIN {X 0,Y 487.811,Z 605.642,A -85,B 0,C 180,E1 -6355.206,E2 -6355.206} C_VEL
LIN {X 0,Y 487.79,Z 605.87,A -85,B 0,C 180,E1 -6355.812,E2 -6355.812} C_VEL
LIN {X 0,Y 487.78,Z 605.668,A -85,B 0,C 180,E1 -6356.803,E2 -6356.803} C_VEL
LIN {X 0,Y 487.85,Z 604.205,A -85,B 0,C 180,E1 -6358.207,E2 -6358.207} C_VEL
LIN {X 0,Y 487.946,Z 602.116,A -85,B 0,C 180,E1 -6359.248,E2 -6359.248} C_VEL
LIN {X 0,Y 487.979,Z 599.327,A -85,B 0,C 180,E1 -6360.237,E2 -6360.237} C_VEL
LIN {X 0,Y 488.086,Z 594.679,A -85,B 0,C 180,E1 -6361.443,E2 -6361.443} C_VEL
LIN {X 0,Y 488.215,Z 590.313,A -85,B 0,C 180,E1 -6362.338,E2 -6362.338} C_VEL
LIN {X 0,Y 488.41,Z 584.328,A -85,B 0,C 180,E1 -6363.331,E2 -6363.331} C_VEL
LIN {X 0,Y 488.586,Z 577.857,A -85,B 0,C 180,E1 -6364.206,E2 -6364.206} C_VEL
LIN {X 0,Y 488.934,Z 568.471,A -85,B 0,C 180,E1 -6365.221,E2 -6365.221} C_VEL
LIN {X 0,Y 489.162,Z 559.9,A -85,B 0,C 180,E1 -6365.941,E2 -6365.941} C_VEL
LIN {X 0,Y 489.41,Z 551.669,A -85,B 0,C 180,E1 -6366.497,E2 -6366.497} C_VEL
LIN {X 0,Y 489.638,Z 542.64,A -85,B 0,C 180,E1 -6366.978,E2 -6366.978} C_VEL
LIN {X 0,Y 489.503,Z 536.461,A -85,B 0,C 180,E1 -6367.247,E2 -6367.247} C_VEL
LIN {X 0,Y 487.998,Z 526.178,A -85,B 0,C 180,E1 -6367.62,E2 -6367.62} C_VEL
LIN {X 0,Y 488.038,Z 519.755,A -85,B 0,C 180,E1 -6370.657,E2 -6370.657} C_VEL
LIN {X 0,Y 488.109,Z 514.234,A -85,B 0,C 180,E1 -6373.263,E2 -6373.263} C_VEL
LIN {X 0,Y 488.173,Z 508.839,A -85,B 0,C 180,E1 -6375.833,E2 -6375.833} C_VEL
LIN {X 0,Y 488.327,Z 503.412,A -85,B 0,C 180,E1 -6378.376,E2 -6378.376} C_VEL
LIN {X 0,Y 488.34,Z 496.21,A -85,B 0,C 180,E1 -6381.725,E2 -6381.725} C_VEL
LIN {X 0,Y 488.373,Z 490.842,A -85,B 0,C 180,E1 -6384.218,E2 -6384.218} C_VEL
LIN {X 0,Y 488.46,Z 487.24,A -85,B 0,C 180,E1 -6385.874,E2 -6385.874} C_VEL
LIN {X 0,Y 488.405,Z 484.462,A -85,B 0,C 180,E1 -6387.216,E2 -6387.216} C_VEL
LIN {X 0,Y 488.889,Z 484.401,A -85,B 0,C 180,E1 -6389.176,E2 -6389.176} C_VEL
LIN {X 0,Y 488.957,Z 484.392,A -85,B 0,C 180,E1 -6390.823,E2 -6390.823} C_VEL
LIN {X 0,Y 488.963,Z 484.392,A -85,B 0,C 180,E1 -6392.471,E2 -6392.471} C_VEL
LIN {X 0,Y 488.859,Z 484.404,A -85,B 0,C 180,E1 -6395.775,E2 -6395.775} C_VEL
LIN {X 0,Y 488.818,Z 484.41,A -85,B 0,C 180,E1 -6398.266,E2 -6398.266} C_VEL
LIN {X 0,Y 488.807,Z 484.411,A -85,B 0,C 180,E1 -6401.612,E2 -6401.612} C_VEL
LIN {X 0,Y 488.766,Z 484.415,A -85,B 0,C 180,E1 -6405,E2 -6405} C_VEL
LIN {X 0,Y 488.756,Z 484.418,A -85,B 0,C 180,E1 -6408.442,E2 -6408.442} C_VEL
LIN {X 0,Y 488.709,Z 484.421,A -85,B 0,C 180,E1 -6411.07,E2 -6411.07} C_VEL
LIN {X 0,Y 488.695,Z 484.425,A -85,B 0,C 180,E1 -6413.745,E2 -6413.745} C_VEL
LIN {X 0,Y 488.799,Z 484.41,A -85,B 0,C 180,E1 -6416.945,E2 -6416.945} C_VEL
LIN {X 0,Y 488.719,Z 484.422,A -85,B 0,C 180,E1 -6420.364,E2 -6420.364} C_VEL
LIN {X 0,Y 488.735,Z 484.419,A -85,B 0,C 180,E1 -6423.484,E2 -6423.484} C_VEL
LIN {X 0,Y 488.689,Z 484.426,A -85,B 0,C 180,E1 -6426.355,E2 -6426.355} C_VEL
LIN {X 0,Y 488.7,Z 484.423,A -85,B 0,C 180,E1 -6429.254,E2 -6429.254} C_VEL
LIN {X 0,Y 488.722,Z 484.421,A -85,B 0,C 180,E1 -6431.602,E2 -6431.602} C_VEL
LIN {X 0,Y 488.711,Z 484.422,A -85,B 0,C 180,E1 -6434.801,E2 -6434.801} C_VEL
LIN {X 0,Y 488.73,Z 484.42,A -85,B 0,C 180,E1 -6437.479,E2 -6437.479} C_VEL
LIN {X 0,Y 488.742,Z 484.418,A -85,B 0,C 180,E1 -6440.75,E2 -6440.75} C_VEL
LIN {X 0,Y 488.675,Z 484.429,A -85,B 0,C 180,E1 -6443.868,E2 -6443.868} C_VEL
LIN {X 0,Y 488.737,Z 484.419,A -85,B 0,C 180,E1 -6446.877,E2 -6446.877} C_VEL
LIN {X 0,Y 488.722,Z 484.423,A -85,B 0,C 180,E1 -6449.781,E2 -6449.781} C_VEL
LIN {X 0,Y 488.797,Z 484.412,A -85,B 0,C 180,E1 -6453.054,E2 -6453.054} C_VEL
LIN {X 0,Y 488.692,Z 484.426,A -85,B 0,C 180,E1 -6456.254,E2 -6456.254} C_VEL
LIN {X 0,Y 488.744,Z 484.419,A -85,B 0,C 180,E1 -6459.175,E2 -6459.175} C_VEL
LIN {X 0,Y 488.757,Z 484.419,A -85,B 0,C 180,E1 -6461.627,E2 -6461.627} C_VEL
LIN {X 0,Y 488.76,Z 484.417,A -85,B 0,C 180,E1 -6464.999,E2 -6464.999} C_VEL
LIN {X 0,Y 488.827,Z 484.41,A -85,B 0,C 180,E1 -6468.388,E2 -6468.388} C_VEL
LIN {X 0,Y 488.816,Z 484.411,A -85,B 0,C 180,E1 -6471.734,E2 -6471.734} C_VEL
LIN {X 0,Y 488.853,Z 484.407,A -85,B 0,C 180,E1 -6474.224,E2 -6474.224} C_VEL
LIN {X 0,Y 488.961,Z 484.392,A -85,B 0,C 180,E1 -6477.529,E2 -6477.529} C_VEL
LIN {X 0,Y 488.968,Z 484.392,A -85,B 0,C 180,E1 -6480,E2 -6480} C_VEL
LIN {X 0,Y 488.959,Z 484.393,A -85,B 0,C 180,E1 -6482.471,E2 -6482.471} C_VEL
LIN {X 0,Y 488.855,Z 484.405,A -85,B 0,C 180,E1 -6485.776,E2 -6485.776} C_VEL
LIN {X 0,Y 488.816,Z 484.411,A -85,B 0,C 180,E1 -6488.266,E2 -6488.266} C_VEL
LIN {X 0,Y 488.803,Z 484.412,A -85,B 0,C 180,E1 -6491.612,E2 -6491.612} C_VEL
LIN {X 0,Y 488.76,Z 484.416,A -85,B 0,C 180,E1 -6495,E2 -6495} C_VEL
LIN {X 0,Y 488.752,Z 484.416,A -85,B 0,C 180,E1 -6498.442,E2 -6498.442} C_VEL
LIN {X 0,Y 488.705,Z 484.423,A -85,B 0,C 180,E1 -6501.071,E2 -6501.071} C_VEL
LIN {X 0,Y 488.692,Z 484.427,A -85,B 0,C 180,E1 -6503.745,E2 -6503.745} C_VEL
LIN {X 0,Y 488.789,Z 484.412,A -85,B 0,C 180,E1 -6506.944,E2 -6506.944} C_VEL
LIN {X 0,Y 488.732,Z 484.419,A -85,B 0,C 180,E1 -6510.219,E2 -6510.219} C_VEL
LIN {X 0,Y 488.733,Z 484.422,A -85,B 0,C 180,E1 -6513.485,E2 -6513.485} C_VEL
LIN {X 0,Y 488.687,Z 484.425,A -85,B 0,C 180,E1 -6516.356,E2 -6516.356} C_VEL
LIN {X 0,Y 488.698,Z 484.426,A -85,B 0,C 180,E1 -6519.254,E2 -6519.254} C_VEL
LIN {X 0,Y 488.721,Z 484.424,A -85,B 0,C 180,E1 -6521.602,E2 -6521.602} C_VEL
LIN {X 0,Y 488.71,Z 484.422,A -85,B 0,C 180,E1 -6524.802,E2 -6524.802} C_VEL
LIN {X 0,Y 488.689,Z 484.428,A -85,B 0,C 180,E1 -6527.475,E2 -6527.475} C_VEL
LIN {X 0,Y 488.747,Z 484.417,A -85,B 0,C 180,E1 -6530.751,E2 -6530.751} C_VEL
LIN {X 0,Y 488.684,Z 484.427,A -85,B 0,C 180,E1 -6533.869,E2 -6533.869} C_VEL
LIN {X 0,Y 488.773,Z 484.528,A -85,B 0,C 180,E1 -6535.935,E2 -6535.935} C_VEL
LIN {X 0,Y 489.853,Z 491.054,A -85,B 0,C 180,E1 -6538.422,E2 -6538.422} C_VEL
LIN {X 0,Y 489.654,Z 497.696,A -85,B 0,C 180,E1 -6540.791,E2 -6540.791} C_VEL
LIN {X 0,Y 489.307,Z 505.679,A -85,B 0,C 180,E1 -6543.561,E2 -6543.561} C_VEL
LIN {X 0,Y 488.991,Z 513.693,A -85,B 0,C 180,E1 -6546.27,E2 -6546.27} C_VEL
LIN {X 0,Y 488.756,Z 522.466,A -85,B 0,C 180,E1 -6549.173,E2 -6549.173} C_VEL
LIN {X 0,Y 488.495,Z 532.502,A -85,B 0,C 180,E1 -6552.415,E2 -6552.415} C_VEL
LIN {X 0,Y 488.288,Z 541.968,A -85,B 0,C 180,E1 -6555.412,E2 -6555.412} C_VEL
LIN {X 0,Y 488.191,Z 551.443,A -85,B 0,C 180,E1 -6558.399,E2 -6558.399} C_VEL
LIN {X 0,Y 489.572,Z 565.247,A -85,B 0,C 180,E1 -6558.878,E2 -6558.878} C_VEL
LIN {X 0,Y 489.355,Z 575.032,A -85,B 0,C 180,E1 -6559.345,E2 -6559.345} C_VEL
LIN {X 0,Y 489.148,Z 583.455,A -85,B 0,C 180,E1 -6559.863,E2 -6559.863} C_VEL
LIN {X 0,Y 488.948,Z 591.594,A -85,B 0,C 180,E1 -6560.486,E2 -6560.486} C_VEL
LIN {X 0,Y 488.644,Z 599.346,A -85,B 0,C 180,E1 -6561.21,E2 -6561.21} C_VEL
LIN {X 0,Y 488.413,Z 607.487,A -85,B 0,C 180,E1 -6562.144,E2 -6562.144} C_VEL
LIN {X 0,Y 488.238,Z 614.648,A -85,B 0,C 180,E1 -6563.18,E2 -6563.18} C_VEL
LIN {X 0,Y 488.152,Z 620.289,A -85,B 0,C 180,E1 -6564.216,E2 -6564.216} C_VEL
LIN {X 0,Y 487.971,Z 625.527,A -85,B 0,C 180,E1 -6565.457,E2 -6565.457} C_VEL
LIN {X 0,Y 488.015,Z 628.219,A -85,B 0,C 180,E1 -6566.285,E2 -6566.285} C_VEL
LIN {X 0,Y 487.935,Z 631.156,A -85,B 0,C 180,E1 -6567.524,E2 -6567.524} C_VEL
LIN {X 0,Y 487.891,Z 632.426,A -85,B 0,C 180,E1 -6568.35,E2 -6568.35} C_VEL
LIN {X 0,Y 487.832,Z 633.208,A -85,B 0,C 180,E1 -6569.175,E2 -6569.175} C_VEL
LIN {X 0,Y 487.816,Z 633.492,A -85,B 0,C 180,E1 -6570,E2 -6570} C_VEL
LIN {X 0,Y 487.832,Z 633.18,A -85,B 0,C 180,E1 -6570.826,E2 -6570.826} C_VEL
LIN {X 0,Y 487.891,Z 632.379,A -85,B 0,C 180,E1 -6571.651,E2 -6571.651} C_VEL
LIN {X 0,Y 487.936,Z 631.089,A -85,B 0,C 180,E1 -6572.477,E2 -6572.477} C_VEL
LIN {X 0,Y 488.018,Z 628.107,A -85,B 0,C 180,E1 -6573.716,E2 -6573.716} C_VEL
LIN {X 0,Y 488.007,Z 623.824,A -85,B 0,C 180,E1 -6574.957,E2 -6574.957} C_VEL
LIN {X 0,Y 488.165,Z 618.621,A -85,B 0,C 180,E1 -6576.082,E2 -6576.082} C_VEL
LIN {X 0,Y 488.293,Z 611.628,A -85,B 0,C 180,E1 -6577.235,E2 -6577.235} C_VEL
LIN {X 0,Y 488.449,Z 605.43,A -85,B 0,C 180,E1 -6578.065,E2 -6578.065} C_VEL
LIN {X 0,Y 488.69,Z 597.906,A -85,B 0,C 180,E1 -6578.894,E2 -6578.894} C_VEL
LIN {X 0,Y 488.934,Z 589.86,A -85,B 0,C 180,E1 -6579.62,E2 -6579.62} C_VEL
LIN {X 0,Y 489.19,Z 579.845,A -85,B 0,C 180,E1 -6580.346,E2 -6580.346} C_VEL
LIN {X 0,Y 489.452,Z 569.234,A -85,B 0,C 180,E1 -6580.916,E2 -6580.916} C_VEL
LIN {X 0,Y 489.335,Z 563.281,A -85,B 0,C 180,E1 -6581.18,E2 -6581.18} C_VEL
LIN {X 0,Y 488.078,Z 551.221,A -85,B 0,C 180,E1 -6581.578,E2 -6581.578} C_VEL
LIN {X 0,Y 488.253,Z 540.671,A -85,B 0,C 180,E1 -6585.017,E2 -6585.017} C_VEL
LIN {X 0,Y 488.401,Z 530.302,A -85,B 0,C 180,E1 -6588.456,E2 -6588.456} C_VEL
LIN {X 0,Y 488.539,Z 522.607,A -85,B 0,C 180,E1 -6591.079,E2 -6591.079} C_VEL
LIN {X 0,Y 488.771,Z 515.058,A -85,B 0,C 180,E1 -6593.742,E2 -6593.742} C_VEL
LIN {X 0,Y 489.092,Z 506.257,A -85,B 0,C 180,E1 -6597.012,E2 -6597.012} C_VEL
LIN {X 0,Y 489.52,Z 498.403,A -85,B 0,C 180,E1 -6600.165,E2 -6600.165} C_VEL
LIN {X 0,Y 489.861,Z 493.835,A -85,B 0,C 180,E1 -6602.171,E2 -6602.171} C_VEL
LIN {X 0,Y 489.665,Z 490.027,A -85,B 0,C 180,E1 -6604.039,E2 -6604.039} C_VEL
LIN {X 0,Y 488.988,Z 485.933,A -85,B 0,C 180,E1 -6606.403,E2 -6606.403} C_VEL
LIN {X 0,Y 488.699,Z 484.426,A -85,B 0,C 180,E1 -6607.439,E2 -6607.439} C_VEL
LIN {X 0,Y 488.72,Z 484.424,A -85,B 0,C 180,E1 -6610.345,E2 -6610.345} C_VEL
LIN {X 0,Y 488.69,Z 484.428,A -85,B 0,C 180,E1 -6613.655,E2 -6613.655} C_VEL
LIN {X 0,Y 488.695,Z 484.427,A -85,B 0,C 180,E1 -6616.347,E2 -6616.347} C_VEL
LIN {X 0,Y 488.722,Z 484.423,A -85,B 0,C 180,E1 -6618.586,E2 -6618.586} C_VEL
LIN {X 0,Y 488.682,Z 484.428,A -85,B 0,C 180,E1 -6621.8,E2 -6621.8} C_VEL
LIN {X 0,Y 488.723,Z 484.423,A -85,B 0,C 180,E1 -6625.053,E2 -6625.053} C_VEL
LIN {X 0,Y 488.675,Z 484.43,A -85,B 0,C 180,E1 -6626.872,E2 -6626.872} C_VEL
LIN {X 0,Y 488.672,Z 485.081,A -85,B 0,C 180,E1 -6628.053,E2 -6628.053} C_VEL
LIN {X 0,Y 488.577,Z 487.81,A -85,B 0,C 180,E1 -6630.72,E2 -6630.72} C_VEL
LIN {X 0,Y 488.453,Z 490.856,A -85,B 0,C 180,E1 -6633.51,E2 -6633.51} C_VEL
LIN {X 0,Y 488.305,Z 493.977,A -85,B 0,C 180,E1 -6636.235,E2 -6636.235} C_VEL
LIN {X 0,Y 488.266,Z 497.625,A -85,B 0,C 180,E1 -6639.326,E2 -6639.326} C_VEL
LIN {X 0,Y 488.126,Z 501.414,A -85,B 0,C 180,E1 -6642.401,E2 -6642.401} C_VEL
LIN {X 0,Y 488.132,Z 504.658,A -85,B 0,C 180,E1 -6644.98,E2 -6644.98} C_VEL
LIN {X 0,Y 488.073,Z 509.278,A -85,B 0,C 180,E1 -6648.545,E2 -6648.545} C_VEL
LIN {X 0,Y 489.591,Z 519.006,A -85,B 0,C 180,E1 -6648.931,E2 -6648.931} C_VEL
LIN {X 0,Y 489.549,Z 527.83,A -85,B 0,C 180,E1 -6649.349,E2 -6649.349} C_VEL
LIN {X 0,Y 489.329,Z 536.414,A -85,B 0,C 180,E1 -6649.867,E2 -6649.867} C_VEL
LIN {X 0,Y 489.118,Z 544.656,A -85,B 0,C 180,E1 -6650.489,E2 -6650.489} C_VEL
LIN {X 0,Y 488.89,Z 552.479,A -85,B 0,C 180,E1 -6651.214,E2 -6651.214} C_VEL
LIN {X 0,Y 488.652,Z 558.949,A -85,B 0,C 180,E1 -6651.939,E2 -6651.939} C_VEL
LIN {X 0,Y 488.477,Z 565.101,A -85,B 0,C 180,E1 -6652.768,E2 -6652.768} C_VEL
LIN {X 0,Y 488.381,Z 571.37,A -85,B 0,C 180,E1 -6653.804,E2 -6653.804} C_VEL
LIN {X 0,Y 488.054,Z 577.22,A -85,B 0,C 180,E1 -6655.044,E2 -6655.044} C_VEL
LIN {X 0,Y 488.132,Z 580.223,A -85,B 0,C 180,E1 -6655.872,E2 -6655.872} C_VEL
LIN {X 0,Y 488,Z 582.565,A -85,B 0,C 180,E1 -6656.698,E2 -6656.698} C_VEL
LIN {X 0,Y 487.994,Z 584.352,A -85,B 0,C 180,E1 -6657.524,E2 -6657.524} C_VEL
LIN {X 0,Y 487.893,Z 585.643,A -85,B 0,C 180,E1 -6658.349,E2 -6658.349} C_VEL
LIN {X 0,Y 487.832,Z 586.453,A -85,B 0,C 180,E1 -6659.175,E2 -6659.175} C_VEL
LIN {X 0,Y 487.817,Z 586.746,A -85,B 0,C 180,E1 -6660,E2 -6660} C_VEL
LIN {X 0,Y 487.833,Z 586.457,A -85,B 0,C 180,E1 -6660.826,E2 -6660.826} C_VEL
LIN {X 0,Y 487.893,Z 585.694,A -85,B 0,C 180,E1 -6661.651,E2 -6661.651} C_VEL
LIN {X 0,Y 487.991,Z 584.455,A -85,B 0,C 180,E1 -6662.476,E2 -6662.476} C_VEL
LIN {X 0,Y 488.036,Z 581.552,A -85,B 0,C 180,E1 -6663.716,E2 -6663.716} C_VEL
LIN {X 0,Y 488.105,Z 578.917,A -85,B 0,C 180,E1 -6664.542,E2 -6664.542} C_VEL
LIN {X 0,Y 488.105,Z 575.659,A -85,B 0,C 180,E1 -6665.37,E2 -6665.37} C_VEL
LIN {X 0,Y 488.416,Z 570.522,A -85,B 0,C 180,E1 -6666.403,E2 -6666.403} C_VEL
LIN {X 0,Y 488.464,Z 564.079,A -85,B 0,C 180,E1 -6667.44,E2 -6667.44} C_VEL
LIN {X 0,Y 488.649,Z 557.74,A -85,B 0,C 180,E1 -6668.269,E2 -6668.269} C_VEL
LIN {X 0,Y 488.993,Z 549.017,A -85,B 0,C 180,E1 -6669.201,E2 -6669.201} C_VEL
LIN {X 0,Y 489.298,Z 538.904,A -85,B 0,C 180,E1 -6670.03,E2 -6670.03} C_VEL
LIN {X 0,Y 489.512,Z 530.972,A -85,B 0,C 180,E1 -6670.548,E2 -6670.548} C_VEL
LIN {X 0,Y 489.649,Z 521.917,A -85,B 0,C 180,E1 -6671.016,E2 -6671.016} C_VEL
LIN {X 0,Y 489.035,Z 514.492,A -85,B 0,C 180,E1 -6671.331,E2 -6671.331} C_VEL
LIN {X 0,Y 488.07,Z 508.3,A -85,B 0,C 180,E1 -6671.56,E2 -6671.56} C_VEL
LIN {X 0,Y 488.07,Z 502.905,A -85,B 0,C 180,E1 -6675.252,E2 -6675.252} C_VEL
LIN {X 0,Y 488.104,Z 498.27,A -85,B 0,C 180,E1 -6678.468,E2 -6678.468} C_VEL
LIN {X 0,Y 488.107,Z 494.54,A -85,B 0,C 180,E1 -6681.098,E2 -6681.098} C_VEL
LIN {X 0,Y 488.134,Z 490.785,A -85,B 0,C 180,E1 -6683.774,E2 -6683.774} C_VEL
LIN {X 0,Y 488.32,Z 486.527,A -85,B 0,C 180,E1 -6686.833,E2 -6686.833} C_VEL
LIN {X 0,Y 488.359,Z 486.161,A -85,B 0,C 180,E1 -6687.252,E2 -6687.252} C_VEL
LIN {X 0,Y 488.372,Z 491.115,A -85,B 0,C 180,E1 -6689.293,E2 -6689.293} C_VEL
LIN {X 0,Y 488.386,Z 497.853,A -85,B 0,C 180,E1 -6692.17,E2 -6692.17} C_VEL
LIN {X 0,Y 488.267,Z 504.755,A -85,B 0,C 180,E1 -6695.152,E2 -6695.152} C_VEL
LIN {X 0,Y 488.198,Z 511.829,A -85,B 0,C 180,E1 -6698.245,E2 -6698.245} C_VEL
LIN {X 0,Y 488.082,Z 517.976,A -85,B 0,C 180,E1 -6700.932,E2 -6700.932} C_VEL
LIN {X 0,Y 488.047,Z 524.305,A -85,B 0,C 180,E1 -6703.726,E2 -6703.726} C_VEL
LIN {X 0,Y 488.077,Z 525.987,A -85,B 0,C 180,E1 -6704.469,E2 -6704.469} C_VEL
LIN {X 0,Y 489.736,Z 537.765,A -85,B 0,C 180,E1 -6704.893,E2 -6704.893} C_VEL
LIN {X 0,Y 489.541,Z 548.173,A -85,B 0,C 180,E1 -6705.384,E2 -6705.384} C_VEL
LIN {X 0,Y 489.255,Z 557.563,A -85,B 0,C 180,E1 -6705.976,E2 -6705.976} C_VEL
LIN {X 0,Y 488.988,Z 565.433,A -85,B 0,C 180,E1 -6706.596,E2 -6706.596} C_VEL
LIN {X 0,Y 488.763,Z 572.893,A -85,B 0,C 180,E1 -6707.315,E2 -6707.315} C_VEL
LIN {X 0,Y 488.519,Z 580.734,A -85,B 0,C 180,E1 -6708.241,E2 -6708.241} C_VEL
LIN {X 0,Y 488.249,Z 588.186,A -85,B 0,C 180,E1 -6709.357,E2 -6709.357} C_VEL
LIN {X 0,Y 488.114,Z 593.813,A -85,B 0,C 180,E1 -6710.446,E2 -6710.446} C_VEL
LIN {X 0,Y 487.994,Z 597.69,A -85,B 0,C 180,E1 -6711.387,E2 -6711.387} C_VEL
LIN {X 0,Y 487.919,Z 601.95,A -85,B 0,C 180,E1 -6712.773,E2 -6712.773} C_VEL
LIN {X 0,Y 487.849,Z 604.055,A -85,B 0,C 180,E1 -6713.796,E2 -6713.796} C_VEL
LIN {X 0,Y 487.819,Z 604.933,A -85,B 0,C 180,E1 -6714.487,E2 -6714.487} C_VEL
LIN {X 0,Y 487.15,Z 605.657,A -85,B 0,C 180,E1 -6715.171,E2 -6715.171} C_VEL
LIN {X 0,Y 484.263,Z 605.988,A -85,B 0,C 180,E1 -6716.289,E2 -6716.289} C_VEL
LIN {X 0,Y 481.39,Z 605.412,A -85,B 0,C 180,E1 -6717.419,E2 -6717.419} C_VEL
LIN {X 0,Y 480.756,Z 604.566,A -85,B 0,C 180,E1 -6718.116,E2 -6718.116} C_VEL
LIN {X 0,Y 480.864,Z 602.461,A -85,B 0,C 180,E1 -6719.233,E2 -6719.233} C_VEL
LIN {X 0,Y 480.886,Z 599.828,A -85,B 0,C 180,E1 -6720.204,E2 -6720.204} C_VEL
LIN {X 0,Y 481.004,Z 596.097,A -85,B 0,C 180,E1 -6721.243,E2 -6721.243} C_VEL
LIN {X 0,Y 481.16,Z 590.869,A -85,B 0,C 180,E1 -6722.36,E2 -6722.36} C_VEL
LIN {X 0,Y 481.334,Z 585.265,A -85,B 0,C 180,E1 -6723.321,E2 -6723.321} C_VEL
LIN {X 0,Y 481.527,Z 578.74,A -85,B 0,C 180,E1 -6724.235,E2 -6724.235} C_VEL
LIN {X 0,Y 481.769,Z 571.287,A -85,B 0,C 180,E1 -6725.088,E2 -6725.088} C_VEL
LIN {X 0,Y 482.146,Z 561.11,A -85,B 0,C 180,E1 -6726.007,E2 -6726.007} C_VEL
LIN {X 0,Y 482.413,Z 552.51,A -85,B 0,C 180,E1 -6726.608,E2 -6726.608} C_VEL
LIN {X 0,Y 482.672,Z 542.868,A -85,B 0,C 180,E1 -6727.133,E2 -6727.133} C_VEL
LIN {X 0,Y 482.393,Z 536.133,A -85,B 0,C 180,E1 -6727.43,E2 -6727.43} C_VEL
LIN {X 0,Y 480.913,Z 526.347,A -85,B 0,C 180,E1 -6727.781,E2 -6727.781} C_VEL
LIN {X 0,Y 480.938,Z 520.928,A -85,B 0,C 180,E1 -6730.36,E2 -6730.36} C_VEL
LIN {X 0,Y 481.019,Z 515.352,A -85,B 0,C 180,E1 -6733.009,E2 -6733.009} C_VEL
